   DATA[746,36] := 1.730048;
   DATA[746,37] := 189.9032;
   DATA[746,38] := 0.000128152;
   DATA[746,39] := 1.0;
   DATA[747,0] := 2.556449;
   DATA[747,1] := 537.959;
   DATA[747,2] := 2.0;
   DATA[747,3] := 1.0;
   DATA[747,4] := 262.1764;
   DATA[747,5] := 8.395475;
   DATA[747,6] := 327.5827;
   DATA[747,7] := 2.323647;
   DATA[747,9] := 1.0;
   DATA[747,10] := 1.0;
   DATA[747,11] := 2.016774;
   DATA[747,13] := 1002.908;
   DATA[747,14] := 1.0;
   DATA[747,15] := 1.0;
   DATA[747,16] := 1.0;
   DATA[747,17] := 1.0;
   DATA[747,18] := 1.0;
   DATA[747,19] := 1.0;
   DATA[747,20] := 148.808;
   DATA[747,21] := 155.8062;
   DATA[747,22] := 1.720309;
   DATA[747,23] := 993.899;
   DATA[747,24] := 2.0;
   DATA[747,25] := 2.0;
   DATA[747,26] := 7.878942;
   DATA[747,27] := 144.7321;
   DATA[747,28] := 263.1056;
   DATA[747,29] := 12.11228;
   DATA[747,30] := 1.731095;
   DATA[747,31] := 1.291789;
   DATA[747,32] := 0.7352687;
   DATA[747,33] := 0.3066329;
   DATA[747,34] := 2.0;
   DATA[747,35] := 251.2977;
   DATA[747,36] := 1.730048;
   DATA[747,37] := 190.0154;
   DATA[747,38] := 0.000128152;
   DATA[747,39] := 1.0;
   DATA[748,0] := 2.536912;
   DATA[748,1] := 538.1553;
   DATA[748,2] := 2.0;
   DATA[748,3] := 1.0;
   DATA[748,4] := 262.1764;
   DATA[748,5] := 8.399321;
   DATA[748,6] := 327.5827;
   DATA[748,7] := 2.09464;
   DATA[748,9] := 1.0;
   DATA[748,10] := 1.0;
   DATA[748,11] := 2.010372;
   DATA[748,13] := 1003.228;
   DATA[748,14] := 1.0;
   DATA[748,15] := 1.0;
   DATA[748,16] := 1.0;
   DATA[748,17] := 1.0;
   DATA[748,18] := 1.0;
   DATA[748,19] := 1.0;
   DATA[748,20] := 148.808;
   DATA[748,21] := 155.8062;
   DATA[748,22] := 1.72159;
   DATA[748,23] := 993.8221;
   DATA[748,24] := 2.0;
   DATA[748,25] := 2.0;
   DATA[748,26] := 7.878942;
   DATA[748,27] := 144.7321;
   DATA[748,28] := 263.1056;
   DATA[748,29] := 12.11228;
   DATA[748,30] := 1.731095;
   DATA[748,31] := 1.288971;
   DATA[748,32] := 0.7352687;
   DATA[748,33] := 0.3066329;
   DATA[748,34] := 2.0;
   DATA[748,35] := 251.2977;
   DATA[748,36] := 1.730048;
   DATA[748,37] := 190.0795;
   DATA[748,38] := 0.000128152;
   DATA[748,39] := 1.0;
   DATA[749,0] := 2.514813;
   DATA[749,1] := 538.5479;
   DATA[749,2] := 2.0;
   DATA[749,3] := 1.0;
   DATA[749,4] := 262.1764;
   DATA[749,5] := 8.399321;
   DATA[749,6] := 327.5827;
   DATA[749,7] := 1.782847;
   DATA[749,9] := 1.0;
   DATA[749,10] := 1.0;
   DATA[749,11] := 2.010372;
   DATA[749,13] := 1003.749;
   DATA[749,14] := 1.0;
   DATA[749,15] := 1.0;
   DATA[749,16] := 1.0;
   DATA[749,17] := 1.0;
   DATA[749,18] := 1.0;
   DATA[749,19] := 1.0;
   DATA[749,20] := 148.808;
   DATA[749,21] := 155.6524;
   DATA[749,22] := 1.721975;
   DATA[749,23] := 993.4376;
   DATA[749,24] := 2.0;
   DATA[749,25] := 2.0;
   DATA[749,26] := 7.878942;
   DATA[749,27] := 144.7321;
   DATA[749,28] := 263.1056;
   DATA[749,29] := 12.11228;
   DATA[749,30] := 1.731095;
   DATA[749,31] := 1.282951;
   DATA[749,32] := 0.7352687;
   DATA[749,33] := 0.3066329;
   DATA[749,34] := 2.0;
   DATA[749,35] := 251.2977;
   DATA[749,36] := 1.730048;
   DATA[749,37] := 190.0795;
   DATA[749,38] := 0.000128152;
   DATA[749,39] := 1.0;
   DATA[750,0] := 2.496237;
   DATA[750,1] := 538.8619;
   DATA[750,2] := 2.0;
   DATA[750,3] := 1.0;
   DATA[750,4] := 262.1764;
   DATA[750,5] := 8.399321;
   DATA[750,6] := 327.5827;
   DATA[750,7] := 1.39365;
   DATA[750,9] := 1.0;
   DATA[750,10] := 1.0;
   DATA[750,11] := 2.010372;
   DATA[750,13] := 1004.31;
   DATA[750,14] := 1.0;
   DATA[750,15] := 1.0;
   DATA[750,16] := 1.0;
   DATA[750,17] := 1.0;
   DATA[750,18] := 1.0;
   DATA[750,19] := 1.0;
   DATA[750,20] := 148.808;
   DATA[750,21] := 155.6524;
   DATA[750,22] := 1.72159;
   DATA[750,23] := 993.6683;
   DATA[750,24] := 2.0;
   DATA[750,25] := 2.0;
   DATA[750,26] := 7.878942;
   DATA[750,27] := 144.7321;
   DATA[750,28] := 263.1056;
   DATA[750,29] := 12.11228;
   DATA[750,30] := 1.731095;
   DATA[750,31] := 1.282439;
   DATA[750,32] := 0.7352687;
   DATA[750,33] := 0.3066329;
   DATA[750,34] := 2.0;
   DATA[750,35] := 251.2977;
   DATA[750,36] := 1.730048;
   DATA[750,37] := 190.0795;
   DATA[750,38] := 0.000128152;
   DATA[750,39] := 1.0;
   DATA[751,0] := 2.480223;
   DATA[751,1] := 538.8226;
   DATA[751,2] := 2.0;
   DATA[751,3] := 1.0;
   DATA[751,4] := 262.1764;
   DATA[751,5] := 8.399321;
   DATA[751,6] := 327.5827;
   DATA[751,7] := 1.022395;
   DATA[751,9] := 1.0;
   DATA[751,10] := 1.0;
   DATA[751,11] := 2.010372;
   DATA[751,13] := 1004.951;
   DATA[751,14] := 1.0;
   DATA[751,15] := 1.0;
   DATA[751,16] := 1.0;
   DATA[751,17] := 1.0;
   DATA[751,18] := 1.0;
   DATA[751,19] := 1.0;
   DATA[751,20] := 148.808;
   DATA[751,21] := 155.6524;
   DATA[751,22] := 1.719668;
   DATA[751,23] := 993.1684;
   DATA[751,24] := 2.0;
   DATA[751,25] := 2.0;
   DATA[751,26] := 7.878942;
   DATA[751,27] := 144.7321;
   DATA[751,28] := 263.1056;
   DATA[751,29] := 12.11228;
   DATA[751,30] := 1.731735;
   DATA[751,31] := 1.281927;
   DATA[751,32] := 0.7352687;
   DATA[751,33] := 0.3066329;
   DATA[751,34] := 2.0;
   DATA[751,35] := 251.2977;
   DATA[751,36] := 1.762086;
   DATA[751,37] := 190.0795;
   DATA[751,38] := 0.000128152;
   DATA[751,39] := 1.0;
   DATA[752,0] := 2.464849;
   DATA[752,1] := 538.9796;
   DATA[752,2] := 2.0;
   DATA[752,3] := 1.0;
   DATA[752,4] := 262.1764;
   DATA[752,5] := 8.399321;
   DATA[752,6] := 327.3263;
   DATA[752,7] := 0.6416557;
   DATA[752,9] := 1.0;
   DATA[752,10] := 1.0;
   DATA[752,11] := 2.010372;
   DATA[752,13] := 1005.351;
   DATA[752,14] := 1.0;
   DATA[752,15] := 1.0;
   DATA[752,16] := 1.0;
   DATA[752,17] := 1.0;
   DATA[752,18] := 1.0;
   DATA[752,19] := 1.0;
   DATA[752,20] := 148.808;
   DATA[752,21] := 155.6524;
   DATA[752,22] := 1.719668;
   DATA[752,23] := 993.1299;
   DATA[752,24] := 2.0;
   DATA[752,25] := 2.0;
   DATA[752,26] := 7.878942;
   DATA[752,27] := 144.7321;
   DATA[752,28] := 263.1056;
   DATA[752,29] := 12.11228;
   DATA[752,30] := 1.734427;
   DATA[752,31] := 1.288075;
   DATA[752,32] := 0.7352687;
   DATA[752,33] := 0.3066329;
   DATA[752,34] := 2.0;
   DATA[752,35] := 251.2977;
   DATA[752,36] := 1.762086;
   DATA[752,37] := 190.0795;
   DATA[752,38] := 0.000128152;
   DATA[752,39] := 1.0;
   DATA[753,0] := 2.449156;
   DATA[753,1] := 539.1759;
   DATA[753,2] := 2.0;
   DATA[753,3] := 1.0;
   DATA[753,4] := 262.1764;
   DATA[753,5] := 8.399321;
   DATA[753,6] := 326.9931;
   DATA[753,7] := 0.3813795;
   DATA[753,8] := 1.0;
   DATA[753,9] := 1.0;
   DATA[753,10] := 1.0;
   DATA[753,11] := 2.010372;
   DATA[753,13] := 1006.272;
   DATA[753,14] := 1.0;
   DATA[753,15] := 1.0;
   DATA[753,16] := 1.0;
   DATA[753,17] := 1.0;
   DATA[753,18] := 1.0;
   DATA[753,19] := 1.0;
   DATA[753,20] := 148.808;
   DATA[753,21] := 155.6524;
   DATA[753,22] := 1.721719;
   DATA[753,23] := 992.361;
   DATA[753,24] := 2.0;
   DATA[753,25] := 2.0;
   DATA[753,26] := 7.878942;
   DATA[753,27] := 144.7321;
   DATA[753,28] := 263.1056;
   DATA[753,29] := 12.11228;
   DATA[753,30] := 1.734427;
   DATA[753,31] := 1.291277;
   DATA[753,32] := 0.7352687;
   DATA[753,33] := 0.3066329;
   DATA[753,34] := 2.0;
   DATA[753,35] := 251.2977;
   DATA[753,36] := 1.762086;
   DATA[753,37] := 190.0795;
   DATA[753,38] := 0.000128152;
   DATA[753,39] := 1.0;
   DATA[754,0] := 2.433462;
   DATA[754,1] := 539.7646;
   DATA[754,2] := 2.0;
   DATA[754,3] := 1.0;
   DATA[754,4] := 262.1764;
   DATA[754,5] := 8.399321;
   DATA[754,6] := 326.7111;
   DATA[754,7] := 0.2296479;
   DATA[754,8] := 1.0;
   DATA[754,9] := 1.0;
   DATA[754,10] := 1.0;
   DATA[754,11] := 2.010372;
   DATA[754,13] := 1006.753;
   DATA[754,14] := 1.0;
   DATA[754,15] := 1.0;
   DATA[754,16] := 1.0;
   DATA[754,17] := 1.0;
   DATA[754,18] := 1.0;
   DATA[754,19] := 1.0;
   DATA[754,20] := 148.808;
   DATA[754,21] := 155.4473;
   DATA[754,22] := 1.721719;
   DATA[754,23] := 992.3225;
   DATA[754,24] := 2.0;
   DATA[754,25] := 2.0;
   DATA[754,26] := 7.878942;
   DATA[754,27] := 144.7321;
   DATA[754,28] := 263.1056;
   DATA[754,29] := 12.11228;
   DATA[754,30] := 1.734427;
   DATA[754,31] := 1.291405;
   DATA[754,32] := 0.7352687;
   DATA[754,33] := 0.3066329;
   DATA[754,34] := 2.0;
   DATA[754,35] := 251.2977;
   DATA[754,36] := 1.762086;
   DATA[754,37] := 190.0795;
   DATA[754,38] := 0.000128152;
   DATA[754,39] := 1.0;
   DATA[755,0] := 2.423213;
   DATA[755,1] := 539.804;
   DATA[755,2] := 2.0;
   DATA[755,3] := 1.0;
   DATA[755,4] := 262.1764;
   DATA[755,5] := 8.399321;
   DATA[755,6] := 326.7111;
   DATA[755,7] := 0.1289206;
   DATA[755,8] := 1.0;
   DATA[755,9] := 1.0;
   DATA[755,10] := 1.0;
   DATA[755,11] := 2.010372;
   DATA[755,13] := 1006.953;
   DATA[755,14] := 1.0;
   DATA[755,15] := 1.0;
   DATA[755,16] := 1.0;
   DATA[755,17] := 1.0;
   DATA[755,18] := 1.0;
   DATA[755,19] := 1.0;
   DATA[755,20] := 148.808;
   DATA[755,21] := 155.4217;
   DATA[755,22] := 1.721719;
   DATA[755,23] := 991.5535;
   DATA[755,24] := 2.0;
   DATA[755,25] := 2.0;
   DATA[755,26] := 7.878942;
   DATA[755,27] := 144.8603;
   DATA[755,28] := 263.1056;
   DATA[755,29] := 12.11228;
   DATA[755,30] := 1.733786;
   DATA[755,31] := 1.291405;
   DATA[755,32] := 0.7352687;
   DATA[755,33] := 0.3066329;
   DATA[755,34] := 2.0;
   DATA[755,35] := 251.2977;
   DATA[755,36] := 1.762086;
   DATA[755,37] := 190.0154;
   DATA[755,38] := 0.000128152;
   DATA[755,39] := 1.0;
   DATA[756,0] := 2.41905;
   DATA[756,1] := 540.3535;
   DATA[756,2] := 2.0;
   DATA[756,3] := 1.0;
   DATA[756,4] := 262.1764;
   DATA[756,5] := 8.399321;
   DATA[756,6] := 326.5573;
   DATA[756,7] := 0.070099;
   DATA[756,8] := 1.0;
   DATA[756,9] := 1.0;
   DATA[756,10] := 1.0;
   DATA[756,11] := 2.010372;
   DATA[756,13] := 1007.474;
   DATA[756,14] := 1.0;
   DATA[756,15] := 1.0;
   DATA[756,16] := 1.0;
   DATA[756,17] := 1.0;
   DATA[756,18] := 1.0;
   DATA[756,19] := 1.0;
   DATA[756,20] := 148.808;
   DATA[756,21] := 155.4217;
   DATA[756,22] := 1.720053;
   DATA[756,23] := 991.7457;
   DATA[756,24] := 2.0;
   DATA[756,25] := 2.0;
   DATA[756,26] := 7.878942;
   DATA[756,27] := 144.8603;
   DATA[756,28] := 263.1056;
   DATA[756,29] := 12.11228;
   DATA[756,30] := 1.731223;
   DATA[756,31] := 1.29243;
   DATA[756,32] := 0.7352687;
   DATA[756,33] := 0.3066329;
   DATA[756,34] := 2.0;
   DATA[756,35] := 251.2977;
   DATA[756,36] := 1.762086;
   DATA[756,37] := 189.8872;
   DATA[756,38] := 0.000128152;
   DATA[756,39] := 1.0;
   DATA[757,0] := 2.41905;
   DATA[757,1] := 540.5497;
   DATA[757,2] := 2.0;
   DATA[757,3] := 1.0;
   DATA[757,4] := 262.1764;
   DATA[757,5] := 8.401243;
   DATA[757,6] := 325.9677;
   DATA[757,7] := 0.03575433;
   DATA[757,8] := 1.0;
   DATA[757,9] := 1.0;
   DATA[757,10] := 1.0;
   DATA[757,11] := 2.010372;
   DATA[757,13] := 1007.835;
   DATA[757,14] := 1.0;
   DATA[757,15] := 1.0;
   DATA[757,16] := 1.0;
   DATA[757,17] := 1.0;
   DATA[757,18] := 1.0;
   DATA[757,19] := 1.0;
   DATA[757,20] := 148.808;
   DATA[757,21] := 155.4217;
   DATA[757,22] := 1.719668;
   DATA[757,23] := 991.3997;
   DATA[757,24] := 2.0;
   DATA[757,25] := 2.0;
   DATA[757,26] := 7.878942;
   DATA[757,27] := 144.8603;
   DATA[757,28] := 263.1056;
   DATA[757,29] := 12.11228;
   DATA[757,30] := 1.731223;
   DATA[757,31] := 1.302165;
   DATA[757,32] := 0.7352687;
   DATA[757,33] := 0.3066329;
   DATA[757,34] := 2.0;
   DATA[757,35] := 251.1535;
   DATA[757,36] := 1.762086;
   DATA[757,37] := 189.8552;
   DATA[757,38] := 0.000128152;
   DATA[757,39] := 1.0;
   DATA[758,0] := 2.437626;
   DATA[758,1] := 541.0992;
   DATA[758,2] := 2.0;
   DATA[758,3] := 1.0;
   DATA[758,4] := 262.1764;
   DATA[758,5] := 8.401243;
   DATA[758,6] := 325.4294;
   DATA[758,7] := 0.01435299;
   DATA[758,8] := 1.0;
   DATA[758,9] := 1.0;
   DATA[758,10] := 1.0;
   DATA[758,11] := 2.010372;
   DATA[758,13] := 1008.355;
   DATA[758,14] := 1.0;
   DATA[758,15] := 1.0;
   DATA[758,16] := 1.0;
   DATA[758,17] := 1.0;
   DATA[758,18] := 1.0;
   DATA[758,19] := 1.0;
   DATA[758,20] := 148.808;
   DATA[758,21] := 155.4217;
   DATA[758,22] := 1.719668;
   DATA[758,23] := 991.3228;
   DATA[758,24] := 2.0;
   DATA[758,25] := 2.0;
   DATA[758,26] := 7.878942;
   DATA[758,27] := 144.8603;
   DATA[758,28] := 263.1056;
   DATA[758,29] := 12.11228;
   DATA[758,30] := 1.731223;
   DATA[758,31] := 1.311387;
   DATA[758,32] := 0.7352687;
   DATA[758,33] := 0.3066329;
   DATA[758,34] := 2.0;
   DATA[758,35] := 251.1055;
   DATA[758,36] := 1.762086;
   DATA[758,37] := 189.8552;
   DATA[758,38] := 0.000128152;
   DATA[758,39] := 1.0;
   DATA[759,0] := 2.461006;
   DATA[759,1] := 540.8245;
   DATA[759,2] := 2.0;
   DATA[759,3] := 1.0;
   DATA[759,4] := 262.1764;
   DATA[759,5] := 8.405088;
   DATA[759,6] := 325.4294;
   DATA[759,7] := 0.000512607;
   DATA[759,8] := 1.0;
   DATA[759,9] := 1.0;
   DATA[759,10] := 1.0;
   DATA[759,11] := 2.010372;
   DATA[759,13] := 1008.275;
   DATA[759,14] := 1.0;
   DATA[759,15] := 1.0;
   DATA[759,16] := 1.0;
   DATA[759,17] := 1.0;
   DATA[759,18] := 1.0;
   DATA[759,19] := 1.0;
   DATA[759,20] := 148.808;
   DATA[759,21] := 155.5242;
   DATA[759,22] := 1.719668;
   DATA[759,23] := 990.4768;
   DATA[759,24] := 2.0;
   DATA[759,25] := 2.0;
   DATA[759,26] := 7.878942;
   DATA[759,27] := 144.8603;
   DATA[759,28] := 263.1056;
   DATA[759,29] := 12.11228;
   DATA[759,30] := 1.731223;
   DATA[759,31] := 1.306648;
   DATA[759,32] := 0.7352687;
   DATA[759,33] := 0.3066329;
   DATA[759,34] := 2.0;
   DATA[759,35] := 251.0734;
   DATA[759,36] := 1.746067;
   DATA[759,37] := 189.8231;
   DATA[759,38] := 0.000128152;
   DATA[759,39] := 1.0;
   DATA[760,0] := 2.478621;
   DATA[760,1] := 541.4918;
   DATA[760,2] := 2.0;
   DATA[760,3] := 1.0;
   DATA[760,4] := 262.1764;
   DATA[760,5] := 8.40605;
   DATA[760,6] := 324.7885;
   DATA[760,7] := 0.000512607;
   DATA[760,8] := 1.0;
   DATA[760,9] := 1.0;
   DATA[760,10] := 1.0;
   DATA[760,11] := 2.010372;
   DATA[760,13] := 1008.355;
   DATA[760,14] := 1.0;
   DATA[760,15] := 1.0;
   DATA[760,16] := 1.0;
   DATA[760,17] := 1.0;
   DATA[760,18] := 1.0;
   DATA[760,19] := 1.0;
   DATA[760,20] := 148.808;
   DATA[760,21] := 155.5242;
   DATA[760,22] := 1.719924;
   DATA[760,23] := 990.3999;
   DATA[760,24] := 2.0;
   DATA[760,25] := 2.0;
   DATA[760,26] := 7.878942;
   DATA[760,27] := 144.8603;
   DATA[760,28] := 263.1056;
   DATA[760,29] := 11.95847;
   DATA[760,30] := 1.731223;
   DATA[760,31] := 1.308185;
   DATA[760,32] := 0.7352687;
   DATA[760,33] := 0.3066329;
   DATA[760,34] := 2.0;
   DATA[760,35] := 250.8652;
   DATA[760,36] := 1.746067;
   DATA[760,37] := 189.727;
   DATA[760,38] := 0.000128152;
   DATA[760,39] := 1.0;
   DATA[761,0] := 2.502642;
   DATA[761,1] := 542.0021;
   DATA[761,2] := 2.0;
   DATA[761,3] := 1.0;
   DATA[761,4] := 262.1764;
   DATA[761,5] := 8.40605;
   DATA[761,6] := 324.1989;
   DATA[761,7] := 0.000512607;
   DATA[761,8] := 1.0;
   DATA[761,9] := 1.0;
   DATA[761,10] := 1.0;
   DATA[761,11] := 2.010372;
   DATA[761,13] := 1008.636;
   DATA[761,14] := 1.0;
   DATA[761,15] := 1.0;
   DATA[761,16] := 1.0;
   DATA[761,17] := 1.0;
   DATA[761,18] := 1.0;
   DATA[761,19] := 1.0;
   DATA[761,20] := 148.808;
   DATA[761,21] := 155.5242;
   DATA[761,22] := 1.719924;
   DATA[761,23] := 990.0154;
   DATA[761,24] := 2.0;
   DATA[761,25] := 2.0;
   DATA[761,26] := 7.878942;
   DATA[761,27] := 144.8603;
   DATA[761,28] := 263.1056;
   DATA[761,29] := 11.95847;
   DATA[761,30] := 1.731223;
   DATA[761,31] := 1.3119;
   DATA[761,32] := 0.7352687;
   DATA[761,33] := 0.3066329;
   DATA[761,34] := 2.0;
   DATA[761,35] := 250.8652;
   DATA[761,36] := 1.746067;
   DATA[761,37] := 189.727;
   DATA[761,38] := 0.000128152;
   DATA[761,39] := 1.0;
   DATA[762,0] := 2.515453;
   DATA[762,1] := 542.3553;
   DATA[762,2] := 2.0;
   DATA[762,3] := 1.0;
   DATA[762,4] := 262.1764;
   DATA[762,5] := 8.408293;
   DATA[762,6] := 323.7375;
   DATA[762,7] := 0.000512607;
   DATA[762,8] := 1.0;
   DATA[762,9] := 1.0;
   DATA[762,10] := 1.0;
   DATA[762,11] := 2.035982;
   DATA[762,13] := 1008.475;
   DATA[762,14] := 1.0;
   DATA[762,15] := 1.0;
   DATA[762,16] := 1.0;
   DATA[762,17] := 1.0;
   DATA[762,18] := 1.0;
   DATA[762,19] := 1.0;
   DATA[762,20] := 148.808;
   DATA[762,21] := 155.5242;
   DATA[762,22] := 1.719924;
   DATA[762,23] := 989.8231;
   DATA[762,24] := 2.0;
   DATA[762,25] := 2.0;
   DATA[762,26] := 7.878942;
   DATA[762,27] := 144.8603;
   DATA[762,28] := 263.1056;
   DATA[762,29] := 11.95847;
   DATA[762,30] := 1.731223;
   DATA[762,31] := 1.304855;
   DATA[762,32] := 0.7352687;
   DATA[762,33] := 0.3066329;
   DATA[762,34] := 2.0;
   DATA[762,35] := 250.8652;
   DATA[762,36] := 1.746067;
   DATA[762,37] := 189.6629;
   DATA[762,38] := 0.000128152;
   DATA[762,39] := 1.0;
   DATA[763,0] := 2.528264;
   DATA[763,1] := 542.9442;
   DATA[763,2] := 2.0;
   DATA[763,3] := 1.0;
   DATA[763,4] := 262.1764;
   DATA[763,5] := 8.412458;
   DATA[763,6] := 323.3017;
   DATA[763,7] := 0.000512607;
   DATA[763,8] := 1.0;
   DATA[763,9] := 1.0;
   DATA[763,10] := 1.0;
   DATA[763,11] := 2.035982;
   DATA[763,13] := 1008.876;
   DATA[763,14] := 1.0;
   DATA[763,15] := 1.0;
   DATA[763,16] := 1.0;
   DATA[763,17] := 1.0;
   DATA[763,18] := 1.0;
   DATA[763,19] := 1.0;
   DATA[763,20] := 148.808;
   DATA[763,21] := 155.5242;
   DATA[763,22] := 1.719924;
   DATA[763,23] := 989.5155;
   DATA[763,24] := 2.0;
   DATA[763,25] := 2.0;
   DATA[763,26] := 7.878942;
   DATA[763,27] := 144.8603;
   DATA[763,28] := 263.1056;
   DATA[763,29] := 11.95847;
   DATA[763,30] := 1.731095;
   DATA[763,31] := 1.291789;
   DATA[763,32] := 0.7352687;
   DATA[763,33] := 0.3066329;
   DATA[763,34] := 2.0;
   DATA[763,35] := 250.8652;
   DATA[763,36] := 1.537821;
   DATA[763,37] := 189.6629;
   DATA[763,38] := 0.000128152;
   DATA[763,39] := 1.0;
   DATA[764,0] := 2.533068;
   DATA[764,1] := 543.4937;
   DATA[764,2] := 2.0;
   DATA[764,3] := 1.0;
   DATA[764,4] := 262.1764;
   DATA[764,5] := 8.412458;
   DATA[764,6] := 323.0197;
   DATA[764,7] := 0.000512607;
   DATA[764,8] := 1.0;
   DATA[764,9] := 1.0;
   DATA[764,10] := 1.0;
   DATA[764,11] := 2.026378;
   DATA[764,13] := 1008.836;
   DATA[764,14] := 1.0;
   DATA[764,15] := 1.0;
   DATA[764,16] := 1.0;
   DATA[764,17] := 1.0;
   DATA[764,18] := 1.0;
   DATA[764,19] := 1.0;
   DATA[764,20] := 148.808;
   DATA[764,21] := 155.5242;
   DATA[764,22] := 1.718771;
   DATA[764,23] := 989.4001;
   DATA[764,24] := 2.0;
   DATA[764,25] := 2.0;
   DATA[764,26] := 7.878942;
   DATA[764,27] := 144.8603;
   DATA[764,28] := 263.1056;
   DATA[764,29] := 11.95847;
   DATA[764,30] := 1.730838;
   DATA[764,31] := 1.28167;
   DATA[764,32] := 0.7352687;
   DATA[764,33] := 0.3066329;
   DATA[764,34] := 2.0;
   DATA[764,35] := 250.8652;
   DATA[764,36] := 1.537821;
   DATA[764,37] := 189.6629;
   DATA[764,38] := 0.000128152;
   DATA[764,39] := 1.0;
   DATA[765,0] := 2.533068;
   DATA[765,1] := 544.0432;
   DATA[765,2] := 2.0;
   DATA[765,3] := 1.0;
   DATA[765,4] := 262.1764;
   DATA[765,5] := 8.412458;
   DATA[765,6] := 322.6096;
   DATA[765,7] := 0.000512607;
   DATA[765,8] := 1.0;
   DATA[765,9] := 1.0;
   DATA[765,10] := 1.0;
   DATA[765,11] := 2.013573;
   DATA[765,13] := 1009.076;
   DATA[765,14] := 1.0;
   DATA[765,15] := 1.0;
   DATA[765,16] := 1.0;
   DATA[765,17] := 1.0;
   DATA[765,18] := 1.0;
   DATA[765,19] := 1.0;
   DATA[765,20] := 148.808;
   DATA[765,21] := 155.5242;
   DATA[765,22] := 1.717233;
   DATA[765,23] := 989.3232;
   DATA[765,24] := 2.0;
   DATA[765,25] := 2.0;
   DATA[765,26] := 7.878942;
   DATA[765,27] := 144.8603;
   DATA[765,28] := 263.1056;
   DATA[765,29] := 11.95847;
   DATA[765,30] := 1.730069;
   DATA[765,31] := 1.28167;
   DATA[765,32] := 0.7352687;
   DATA[765,33] := 0.3066329;
   DATA[765,34] := 2.0;
   DATA[765,35] := 250.8652;
   DATA[765,36] := 1.665972;
   DATA[765,37] := 189.5828;
   DATA[765,38] := 0.000128152;
   DATA[765,39] := 1.0;
   DATA[766,0] := 2.533068;
   DATA[766,1] := 544.7498;
   DATA[766,2] := 2.0;
   DATA[766,3] := 1.0;
   DATA[766,4] := 262.1764;
   DATA[766,5] := 8.417906;
   DATA[766,6] := 321.8405;
   DATA[766,7] := 0.000512607;
   DATA[766,8] := 1.0;
   DATA[766,9] := 1.0;
   DATA[766,10] := 1.0;
   DATA[766,11] := 2.013573;
   DATA[766,13] := 1008.916;
   DATA[766,14] := 1.0;
   DATA[766,15] := 1.0;
   DATA[766,16] := 1.0;
   DATA[766,17] := 1.0;
   DATA[766,18] := 1.0;
   DATA[766,19] := 1.0;
   DATA[766,20] := 148.808;
   DATA[766,21] := 155.5242;
   DATA[766,22] := 1.717233;
   DATA[766,23] := 989.2848;
   DATA[766,24] := 2.0;
   DATA[766,25] := 2.0;
   DATA[766,26] := 7.878942;
   DATA[766,27] := 144.8603;
   DATA[766,28] := 263.1056;
   DATA[766,29] := 11.95847;
   DATA[766,30] := 1.728275;
   DATA[766,31] := 1.28167;
   DATA[766,32] := 0.7352687;
   DATA[766,33] := 0.3066329;
   DATA[766,34] := 2.0;
   DATA[766,35] := 250.8652;
   DATA[766,36] := 1.69801;
   DATA[766,37] := 189.5828;
   DATA[766,38] := 0.000128152;
   DATA[766,39] := 1.0;
   DATA[767,0] := 2.531467;
   DATA[767,1] := 545.4563;
   DATA[767,2] := 2.0;
   DATA[767,3] := 1.0;
   DATA[767,4] := 262.1764;
   DATA[767,5] := 8.422392;
   DATA[767,6] := 321.4048;
   DATA[767,8] := 1.0;
   DATA[767,9] := 1.0;
   DATA[767,10] := 1.0;
   DATA[767,11] := 2.013573;
   DATA[767,13] := 1009.637;
   DATA[767,14] := 1.0;
   DATA[767,15] := 1.0;
   DATA[767,16] := 1.0;
   DATA[767,17] := 1.0;
   DATA[767,18] := 1.0;
   DATA[767,19] := 1.0;
   DATA[767,20] := 148.808;
   DATA[767,21] := 155.5242;
   DATA[767,22] := 1.717233;
   DATA[767,23] := 988.5157;
   DATA[767,24] := 2.0;
   DATA[767,25] := 2.0;
   DATA[767,26] := 7.878942;
   DATA[767,27] := 144.8603;
   DATA[767,28] := 263.1056;
   DATA[767,29] := 11.95847;
   DATA[767,30] := 1.728275;
   DATA[767,31] := 1.294479;
   DATA[767,32] := 0.7352687;
   DATA[767,33] := 0.3066329;
   DATA[767,34] := 2.0;
   DATA[767,35] := 250.7049;
   DATA[767,36] := 1.69801;
   DATA[767,37] := 189.4066;
   DATA[767,38] := 0.000128152;
   DATA[767,39] := 1.0;
   DATA[768,0] := 2.531467;
   DATA[768,1] := 546.3199;
   DATA[768,2] := 2.0;
   DATA[768,3] := 1.0;
   DATA[768,4] := 262.1764;
   DATA[768,5] := 8.422712;
   DATA[768,6] := 320.8665;
   DATA[768,8] := 1.0;
   DATA[768,9] := 1.0;
   DATA[768,10] := 1.0;
   DATA[768,11] := 2.013573;
   DATA[768,13] := 1009.637;
   DATA[768,14] := 1.0;
   DATA[768,15] := 1.0;
   DATA[768,16] := 1.0;
   DATA[768,17] := 1.0;
   DATA[768,18] := 1.0;
   DATA[768,19] := 1.0;
   DATA[768,20] := 148.808;
   DATA[768,21] := 155.5242;
   DATA[768,22] := 1.717233;
   DATA[768,23] := 988.0543;
   DATA[768,24] := 2.0;
   DATA[768,25] := 2.0;
   DATA[768,26] := 7.878942;
   DATA[768,27] := 144.8603;
   DATA[768,28] := 263.1056;
   DATA[768,29] := 11.95847;
   DATA[768,30] := 1.728275;
   DATA[768,31] := 1.294479;
   DATA[768,32] := 0.7352687;
   DATA[768,33] := 0.3066329;
   DATA[768,34] := 2.0;
   DATA[768,35] := 250.6248;
   DATA[768,36] := 1.69801;
   DATA[768,37] := 189.3265;
   DATA[768,38] := 0.000128152;
   DATA[768,39] := 1.0;
   DATA[769,0] := 2.531467;
   DATA[769,1] := 546.4376;
   DATA[769,2] := 2.0;
   DATA[769,3] := 1.0;
   DATA[769,4] := 262.1764;
   DATA[769,5] := 8.425276;
   DATA[769,6] := 320.687;
   DATA[769,8] := 1.0;
   DATA[769,9] := 1.0;
   DATA[769,10] := 1.0;
   DATA[769,11] := 2.013573;
   DATA[769,13] := 1009.917;
   DATA[769,14] := 1.0;
   DATA[769,15] := 1.0;
   DATA[769,16] := 1.0;
   DATA[769,17] := 1.0;
   DATA[769,18] := 1.0;
   DATA[769,19] := 1.0;
   DATA[769,20] := 148.808;
   DATA[769,21] := 155.5242;
   DATA[769,22] := 1.717233;
   DATA[769,23] := 987.5544;
   DATA[769,24] := 2.0;
   DATA[769,25] := 2.0;
   DATA[769,26] := 7.878942;
   DATA[769,27] := 144.9116;
   DATA[769,28] := 263.1056;
   DATA[769,29] := 11.95847;
   DATA[769,30] := 1.728275;
   DATA[769,31] := 1.291533;
   DATA[769,32] := 0.7352687;
   DATA[769,33] := 0.3074016;
   DATA[769,34] := 2.0;
   DATA[769,35] := 250.6248;
   DATA[769,36] := 1.69801;
   DATA[769,37] := 189.3265;
   DATA[769,38] := 0.000128152;
   DATA[769,39] := 1.0;
   DATA[770,0] := 2.53435;
   DATA[770,1] := 546.6732;
   DATA[770,2] := 2.0;
   DATA[770,3] := 1.0;
   DATA[770,4] := 262.1764;
   DATA[770,5] := 8.432005;
   DATA[770,6] := 320.2512;
   DATA[770,8] := 1.0;
   DATA[770,9] := 1.0;
   DATA[770,10] := 1.0;
   DATA[770,11] := 2.013573;
   DATA[770,13] := 1009.877;
   DATA[770,14] := 1.0;
   DATA[770,15] := 1.0;
   DATA[770,16] := 1.0;
   DATA[770,17] := 1.0;
   DATA[770,18] := 1.0;
   DATA[770,19] := 1.0;
   DATA[770,20] := 148.808;
   DATA[770,21] := 155.5242;
   DATA[770,22] := 1.715952;
   DATA[770,23] := 987.1315;
   DATA[770,24] := 2.0;
   DATA[770,25] := 2.0;
   DATA[770,26] := 7.878942;
   DATA[770,27] := 144.9628;
   DATA[770,28] := 263.1056;
   DATA[770,29] := 11.95847;
   DATA[770,30] := 1.728275;
   DATA[770,31] := 1.290765;
   DATA[770,32] := 0.7352687;
   DATA[770,33] := 0.3074016;
   DATA[770,34] := 2.0;
   DATA[770,35] := 250.785;
   DATA[770,36] := 1.69801;
   DATA[770,37] := 189.5027;
   DATA[770,38] := 0.000128152;
   DATA[770,39] := 1.0;
   DATA[771,0] := 2.53435;
   DATA[771,1] := 546.6732;
   DATA[771,2] := 2.0;
   DATA[771,3] := 1.0;
   DATA[771,4] := 262.1764;
   DATA[771,5] := 8.432005;
   DATA[771,6] := 320.2512;
   DATA[771,8] := 1.0;
   DATA[771,9] := 1.0;
   DATA[771,10] := 1.0;
   DATA[771,11] := 2.013573;
   DATA[771,13] := 1009.877;
   DATA[771,14] := 1.0;
   DATA[771,15] := 1.0;
   DATA[771,16] := 1.0;
   DATA[771,17] := 1.0;
   DATA[771,18] := 1.0;
   DATA[771,19] := 1.0;
   DATA[771,20] := 148.808;
   DATA[771,21] := 155.5242;
   DATA[771,22] := 1.715952;
   DATA[771,23] := 987.1315;
   DATA[771,24] := 2.0;
   DATA[771,25] := 2.0;
   DATA[771,26] := 7.878942;
   DATA[771,27] := 144.9628;
   DATA[771,28] := 263.1056;
   DATA[771,29] := 11.95847;
   DATA[771,30] := 1.728275;
   DATA[771,31] := 1.290765;
   DATA[771,32] := 0.7352687;
   DATA[771,33] := 0.3074016;
   DATA[771,34] := 2.0;
   DATA[771,35] := 250.785;
   DATA[771,36] := 1.69801;
   DATA[771,37] := 189.5027;
   DATA[771,38] := 0.000128152;
   DATA[771,39] := 1.0;
   DATA[772,0] := 2.537232;
   DATA[772,1] := 546.5947;
   DATA[772,2] := 2.0;
   DATA[772,3] := 1.0;
   DATA[772,4] := 262.1764;
   DATA[772,5] := 8.432005;
   DATA[772,6] := 319.5847;
   DATA[772,8] := 1.0;
   DATA[772,9] := 1.0;
   DATA[772,10] := 1.0;
   DATA[772,11] := 2.013573;
   DATA[772,13] := 1010.038;
   DATA[772,14] := 1.0;
   DATA[772,15] := 1.0;
   DATA[772,16] := 1.0;
   DATA[772,17] := 1.0;
   DATA[772,18] := 1.0;
   DATA[772,19] := 1.0;
   DATA[772,20] := 148.808;
   DATA[772,21] := 155.5242;
   DATA[772,22] := 1.715952;
   DATA[772,23] := 986.747;
   DATA[772,24] := 2.0;
   DATA[772,25] := 2.0;
   DATA[772,26] := 7.878942;
   DATA[772,27] := 144.9628;
   DATA[772,28] := 263.1056;
   DATA[772,29] := 11.95847;
   DATA[772,30] := 1.728275;
   DATA[772,31] := 1.282183;
   DATA[772,32] := 0.7352687;
   DATA[772,33] := 0.3074016;
   DATA[772,34] := 2.0;
   DATA[772,35] := 250.9613;
   DATA[772,36] := 1.69801;
   DATA[772,37] := 189.6949;
   DATA[772,38] := 0.000128152;
   DATA[772,39] := 1.0;
   DATA[773,0] := 2.537232;
   DATA[773,1] := 546.6339;
   DATA[773,2] := 2.0;
   DATA[773,3] := 1.0;
   DATA[773,4] := 262.1764;
   DATA[773,5] := 8.434568;
   DATA[773,6] := 319.5847;
   DATA[773,8] := 1.0;
   DATA[773,9] := 1.0;
   DATA[773,10] := 1.0;
   DATA[773,11] := 2.013573;
   DATA[773,13] := 1009.917;
   DATA[773,14] := 1.0;
   DATA[773,15] := 1.0;
   DATA[773,16] := 1.0;
   DATA[773,17] := 1.0;
   DATA[773,18] := 1.0;
   DATA[773,19] := 1.0;
   DATA[773,20] := 148.808;
   DATA[773,21] := 155.5242;
   DATA[773,22] := 1.715952;
   DATA[773,23] := 986.2087;
   DATA[773,24] := 2.0;
   DATA[773,25] := 2.0;
   DATA[773,26] := 7.878942;
   DATA[773,27] := 144.9628;
   DATA[773,28] := 263.1056;
   DATA[773,29] := 11.95847;
   DATA[773,30] := 1.728788;
   DATA[773,31] := 1.290252;
   DATA[773,32] := 0.7352687;
   DATA[773,33] := 0.3065048;
   DATA[773,34] := 2.0;
   DATA[773,35] := 250.9613;
   DATA[773,36] := 1.649953;
   DATA[773,37] := 189.759;
   DATA[773,38] := 0.000128152;
   DATA[773,39] := 1.0;
   DATA[774,0] := 2.537232;
   DATA[774,1] := 547.0264;
   DATA[774,2] := 2.0;
   DATA[774,3] := 1.0;
   DATA[774,4] := 262.1764;
   DATA[774,5] := 8.439695;
   DATA[774,6] := 318.9695;
   DATA[774,8] := 1.0;
   DATA[774,9] := 1.0;
   DATA[774,10] := 1.0;
   DATA[774,11] := 2.013573;
   DATA[774,13] := 1009.757;
   DATA[774,14] := 1.0;
   DATA[774,15] := 1.0;
   DATA[774,16] := 1.0;
   DATA[774,17] := 1.0;
   DATA[774,18] := 1.0;
   DATA[774,19] := 1.0;
   DATA[774,20] := 148.808;
   DATA[774,21] := 155.6524;
   DATA[774,22] := 1.717746;
   DATA[774,23] := 986.0164;
   DATA[774,24] := 2.0;
   DATA[774,25] := 2.0;
   DATA[774,26] := 7.878942;
   DATA[774,27] := 144.9628;
   DATA[774,28] := 263.1056;
   DATA[774,29] := 11.95847;
   DATA[774,30] := 1.731864;
   DATA[774,31] := 1.297554;
   DATA[774,32] := 0.7352687;
   DATA[774,33] := 0.3065048;
   DATA[774,34] := 2.0;
   DATA[774,35] := 250.9613;
   DATA[774,36] := 1.649953;
   DATA[774,37] := 189.759;
   DATA[774,38] := 0.000128152;
   DATA[774,39] := 1.0;
   DATA[775,0] := 2.537232;
   DATA[775,1] := 546.9872;
   DATA[775,2] := 2.0;
   DATA[775,3] := 1.0;
   DATA[775,4] := 262.1764;
   DATA[775,5] := 8.4429;
   DATA[775,6] := 318.9695;
   DATA[775,8] := 1.0;
   DATA[775,9] := 1.0;
   DATA[775,10] := 1.0;
   DATA[775,11] := 2.013573;
   DATA[775,13] := 1010.078;
   DATA[775,14] := 1.0;
   DATA[775,15] := 1.0;
   DATA[775,16] := 1.0;
   DATA[775,17] := 1.0;
   DATA[775,18] := 1.0;
   DATA[775,19] := 1.0;
   DATA[775,20] := 148.808;
   DATA[775,21] := 155.6524;
   DATA[775,22] := 1.717746;
   DATA[775,23] := 985.5934;
   DATA[775,24] := 2.0;
   DATA[775,25] := 2.0;
   DATA[775,26] := 7.878942;
   DATA[775,27] := 144.9628;
   DATA[775,28] := 263.1056;
   DATA[775,29] := 11.95847;
   DATA[775,30] := 1.731864;
   DATA[775,31] := 1.308569;
   DATA[775,32] := 0.7352687;
   DATA[775,33] := 0.3065048;
   DATA[775,34] := 2.0;
   DATA[775,35] := 250.9613;
   DATA[775,36] := 1.649953;
   DATA[775,37] := 189.759;
   DATA[775,38] := 0.000128152;
   DATA[775,39] := 1.0;
   DATA[776,0] := 2.537232;
   DATA[776,1] := 546.8694;
   DATA[776,2] := 2.0;
   DATA[776,3] := 1.0;
   DATA[776,4] := 262.1764;
   DATA[776,5] := 8.4429;
   DATA[776,6] := 318.8926;
   DATA[776,8] := 1.0;
   DATA[776,9] := 1.0;
   DATA[776,10] := 1.0;
   DATA[776,11] := 2.013573;
   DATA[776,13] := 1010.638;
   DATA[776,14] := 1.0;
   DATA[776,15] := 1.0;
   DATA[776,16] := 1.0;
   DATA[776,17] := 1.0;
   DATA[776,18] := 1.0;
   DATA[776,19] := 1.0;
   DATA[776,20] := 148.808;
   DATA[776,21] := 155.7293;
   DATA[776,22] := 1.717746;
   DATA[776,23] := 985.2089;
   DATA[776,24] := 2.0;
   DATA[776,25] := 2.0;
   DATA[776,26] := 7.878942;
   DATA[776,27] := 144.9628;
   DATA[776,28] := 263.1056;
   DATA[776,29] := 11.95847;
   DATA[776,30] := 1.731864;
   DATA[776,31] := 1.318432;
   DATA[776,32] := 0.7352687;
   DATA[776,33] := 0.3065048;
   DATA[776,34] := 2.0;
   DATA[776,35] := 250.9613;
   DATA[776,36] := 1.649953;
   DATA[776,37] := 189.759;
   DATA[776,38] := 0.000128152;
   DATA[776,39] := 1.0;
   DATA[777,0] := 2.542677;
   DATA[777,1] := 547.262;
   DATA[777,2] := 2.0;
   DATA[777,3] := 1.0;
   DATA[777,4] := 262.1764;
   DATA[777,5] := 8.444822;
   DATA[777,6] := 318.3799;
   DATA[777,8] := 1.0;
   DATA[777,9] := 1.0;
   DATA[777,10] := 1.0;
   DATA[777,11] := 2.013573;
   DATA[777,13] := 1010.839;
   DATA[777,14] := 1.0;
   DATA[777,15] := 1.0;
   DATA[777,16] := 1.0;
   DATA[777,17] := 1.0;
   DATA[777,18] := 1.0;
   DATA[777,19] := 1.0;
   DATA[777,20] := 148.808;
   DATA[777,21] := 155.7293;
   DATA[777,22] := 1.717361;
   DATA[777,23] := 984.5937;
   DATA[777,24] := 2.0;
   DATA[777,25] := 2.0;
   DATA[777,26] := 7.878942;
   DATA[777,27] := 144.9628;
   DATA[777,28] := 263.1056;
   DATA[777,29] := 11.95847;
   DATA[777,30] := 1.731864;
   DATA[777,31] := 1.321506;
   DATA[777,32] := 0.7352687;
   DATA[777,33] := 0.3065048;
   DATA[777,34] := 2.0;
   DATA[777,35] := 251.1055;
   DATA[777,36] := 1.649953;
   DATA[777,37] := 189.759;
   DATA[777,38] := 0.000128152;
   DATA[777,39] := 1.0;
   DATA[778,0] := 2.543958;
   DATA[778,1] := 547.6152;
   DATA[778,2] := 2.0;
   DATA[778,3] := 1.0;
   DATA[778,4] := 262.1764;
   DATA[778,5] := 8.449949;
   DATA[778,6] := 318.2774;
   DATA[778,8] := 1.0;
   DATA[778,9] := 1.0;
   DATA[778,10] := 1.0;
   DATA[778,11] := 2.013573;
   DATA[778,13] := 1010.758;
   DATA[778,14] := 1.0;
   DATA[778,15] := 1.0;
   DATA[778,16] := 1.0;
   DATA[778,17] := 1.0;
   DATA[778,18] := 1.0;
   DATA[778,19] := 1.0;
   DATA[778,20] := 148.808;
   DATA[778,21] := 155.7293;
   DATA[778,22] := 1.717233;
   DATA[778,23] := 984.4014;
   DATA[778,24] := 2.0;
   DATA[778,25] := 2.0;
   DATA[778,26] := 7.878942;
   DATA[778,27] := 144.9628;
   DATA[778,28] := 263.1056;
   DATA[778,29] := 11.95847;
   DATA[778,30] := 1.731864;
   DATA[778,31] := 1.31254;
   DATA[778,32] := 0.7352687;
   DATA[778,33] := 0.3065048;
   DATA[778,34] := 2.0;
   DATA[778,35] := 251.1055;
   DATA[778,36] := 1.649953;
   DATA[778,37] := 189.759;
   DATA[778,38] := 0.000128152;
   DATA[778,39] := 1.0;
   DATA[779,0] := 2.543958;
   DATA[779,1] := 547.4975;
   DATA[779,2] := 2.0;
   DATA[779,3] := 1.0;
   DATA[779,4] := 262.1764;
   DATA[779,5] := 8.452192;
   DATA[779,6] := 317.9954;
   DATA[779,8] := 1.0;
   DATA[779,9] := 1.0;
   DATA[779,10] := 1.0;
   DATA[779,11] := 2.013573;
   DATA[779,13] := 1010.758;
   DATA[779,14] := 1.0;
   DATA[779,15] := 1.0;
   DATA[779,16] := 1.0;
   DATA[779,17] := 1.0;
   DATA[779,18] := 1.0;
   DATA[779,19] := 1.0;
   DATA[779,20] := 148.808;
   DATA[779,21] := 155.7293;
   DATA[779,22] := 1.717233;
   DATA[779,23] := 983.7862;
   DATA[779,24] := 2.0;
   DATA[779,25] := 2.0;
   DATA[779,26] := 7.878942;
   DATA[779,27] := 144.9628;
   DATA[779,28] := 263.1056;
   DATA[779,29] := 11.95847;
   DATA[779,30] := 1.731864;
   DATA[779,31] := 1.304214;
   DATA[779,32] := 0.7352687;
   DATA[779,33] := 0.3065048;
   DATA[779,34] := 2.0;
   DATA[779,35] := 251.1055;
   DATA[779,36] := 1.649953;
   DATA[779,37] := 189.759;
   DATA[779,38] := 0.000128152;
   DATA[779,39] := 1.0;
   DATA[780,0] := 2.543958;
   DATA[780,1] := 547.4582;
   DATA[780,2] := 2.0;
   DATA[780,3] := 1.0;
   DATA[780,4] := 262.1764;
   DATA[780,5] := 8.452833;
   DATA[780,6] := 317.9185;
   DATA[780,8] := 1.0;
   DATA[780,9] := 1.0;
   DATA[780,10] := 1.0;
   DATA[780,11] := 2.013573;
   DATA[780,13] := 1010.638;
   DATA[780,14] := 1.0;
   DATA[780,15] := 1.0;
   DATA[780,16] := 1.0;
   DATA[780,17] := 1.0;
   DATA[780,18] := 1.0;
   DATA[780,19] := 1.0;
   DATA[780,20] := 148.808;
   DATA[780,21] := 155.7293;
   DATA[780,22] := 1.717233;
   DATA[780,23] := 983.5939;
   DATA[780,24] := 2.0;
   DATA[780,25] := 2.0;
   DATA[780,26] := 7.878942;
   DATA[780,27] := 144.9628;
   DATA[780,28] := 263.1056;
   DATA[780,29] := 11.95847;
   DATA[780,30] := 1.730582;
   DATA[780,31] := 1.297682;
   DATA[780,32] := 0.7352687;
   DATA[780,33] := 0.3065048;
   DATA[780,34] := 2.0;
   DATA[780,35] := 251.1055;
   DATA[780,36] := 1.649953;
   DATA[780,37] := 189.759;
   DATA[780,38] := 0.000128152;
   DATA[780,39] := 1.0;
   DATA[781,0] := 2.539474;
   DATA[781,1] := 547.4189;
   DATA[781,2] := 2.0;
   DATA[781,3] := 1.0;
   DATA[781,4] := 262.1764;
   DATA[781,5] := 8.452833;
   DATA[781,6] := 317.8672;
   DATA[781,8] := 1.0;
   DATA[781,9] := 1.0;
   DATA[781,10] := 1.0;
   DATA[781,11] := 2.013573;
   DATA[781,13] := 1010.758;
   DATA[781,14] := 1.0;
   DATA[781,15] := 1.0;
   DATA[781,16] := 1.0;
   DATA[781,17] := 1.0;
   DATA[781,18] := 1.0;
   DATA[781,19] := 1.0;
   DATA[781,20] := 148.808;
   DATA[781,21] := 155.7293;
   DATA[781,22] := 1.717233;
   DATA[781,23] := 983.0556;
   DATA[781,24] := 2.0;
   DATA[781,25] := 2.0;
   DATA[781,26] := 7.878942;
   DATA[781,27] := 144.9628;
   DATA[781,28] := 263.1056;
   DATA[781,29] := 11.95847;
   DATA[781,30] := 1.730582;
   DATA[781,31] := 1.291533;
   DATA[781,32] := 0.7352687;
   DATA[781,33] := 0.3065048;
   DATA[781,34] := 2.0;
   DATA[781,35] := 251.1055;
   DATA[781,36] := 1.69801;
   DATA[781,37] := 189.759;
   DATA[781,38] := 0.000128152;
   DATA[781,39] := 1.0;
   DATA[782,0] := 2.537873;
   DATA[782,1] := 547.9685;
   DATA[782,2] := 2.0;
   DATA[782,3] := 1.0;
   DATA[782,4] := 262.1764;
   DATA[782,5] := 8.456038;
   DATA[782,6] := 317.7903;
   DATA[782,8] := 1.0;
   DATA[782,9] := 1.0;
   DATA[782,10] := 1.0;
   DATA[782,11] := 2.042384;
   DATA[782,13] := 1010.438;
   DATA[782,14] := 1.0;
   DATA[782,15] := 1.0;
   DATA[782,16] := 1.0;
   DATA[782,17] := 1.0;
   DATA[782,18] := 1.0;
   DATA[782,19] := 1.0;
   DATA[782,20] := 148.808;
   DATA[782,21] := 155.7293;
   DATA[782,22] := 1.717233;
   DATA[782,23] := 982.4789;
   DATA[782,24] := 2.0;
   DATA[782,25] := 2.0;
   DATA[782,26] := 7.878942;
   DATA[782,27] := 144.9628;
   DATA[782,28] := 263.1056;
   DATA[782,29] := 11.95847;
   DATA[782,30] := 1.730582;
   DATA[782,31] := 1.291533;
   DATA[782,32] := 0.7352687;
   DATA[782,33] := 0.3065048;
   DATA[782,34] := 2.0;
   DATA[782,35] := 251.1055;
   DATA[782,36] := 1.69801;
   DATA[782,37] := 189.759;
   DATA[782,38] := 0.000128152;
   DATA[782,39] := 1.0;
   DATA[783,0] := 2.537873;
   DATA[783,1] := 548.9891;
   DATA[783,2] := 2.0;
   DATA[783,3] := 1.0;
   DATA[783,4] := 262.1764;
   DATA[783,5] := 8.456038;
   DATA[783,6] := 317.6109;
   DATA[783,8] := 1.0;
   DATA[783,9] := 1.0;
   DATA[783,10] := 1.0;
   DATA[783,11] := 2.042384;
   DATA[783,13] := 1010.518;
   DATA[783,14] := 1.0;
   DATA[783,15] := 1.0;
   DATA[783,16] := 1.0;
   DATA[783,17] := 1.0;
   DATA[783,18] := 1.0;
   DATA[783,19] := 1.0;
   DATA[783,20] := 148.808;
   DATA[783,21] := 155.7293;
   DATA[783,22] := 1.720309;
   DATA[783,23] := 982.4404;
   DATA[783,24] := 2.0;
   DATA[783,25] := 2.0;
   DATA[783,26] := 7.878942;
   DATA[783,27] := 144.9628;
   DATA[783,28] := 263.1056;
   DATA[783,29] := 11.95847;
   DATA[783,30] := 1.728788;
   DATA[783,31] := 1.295888;
   DATA[783,32] := 0.7352687;
   DATA[783,33] := 0.3065048;
   DATA[783,34] := 2.0;
   DATA[783,35] := 251.1055;
   DATA[783,36] := 1.69801;
   DATA[783,37] := 189.759;
   DATA[783,38] := 0.000128152;
   DATA[783,39] := 1.0;
   DATA[784,0] := 2.533709;
   DATA[784,1] := 549.7349;
   DATA[784,2] := 2.0;
   DATA[784,3] := 1.0;
   DATA[784,4] := 262.1764;
   DATA[784,5] := 8.456038;
   DATA[784,6] := 317.5083;
   DATA[784,8] := 1.0;
   DATA[784,9] := 1.0;
   DATA[784,10] := 1.0;
   DATA[784,11] := 2.042384;
   DATA[784,13] := 1010.678;
   DATA[784,14] := 1.0;
   DATA[784,15] := 1.0;
   DATA[784,16] := 1.0;
   DATA[784,17] := 1.0;
   DATA[784,18] := 1.0;
   DATA[784,19] := 1.0;
   DATA[784,20] := 148.808;
   DATA[784,21] := 155.7293;
   DATA[784,22] := 1.720309;
   DATA[784,23] := 982.2482;
   DATA[784,24] := 2.0;
   DATA[784,25] := 2.0;
   DATA[784,26] := 7.878942;
   DATA[784,27] := 144.9628;
   DATA[784,28] := 263.1056;
   DATA[784,29] := 11.95847;
   DATA[784,30] := 1.728788;
   DATA[784,31] := 1.291405;
   DATA[784,32] := 0.7352687;
   DATA[784,33] := 0.3065048;
   DATA[784,34] := 2.0;
   DATA[784,35] := 250.9613;
   DATA[784,36] := 1.69801;
   DATA[784,37] := 189.759;
   DATA[784,38] := 0.000128152;
   DATA[784,39] := 1.0;
   DATA[785,0] := 2.533709;
   DATA[785,1] := 549.6564;
   DATA[785,2] := 2.0;
   DATA[785,3] := 1.0;
   DATA[785,4] := 262.1764;
   DATA[785,5] := 8.45764;
   DATA[785,6] := 317.252;
   DATA[785,8] := 1.0;
   DATA[785,9] := 1.0;
   DATA[785,10] := 1.0;
   DATA[785,11] := 2.042384;
   DATA[785,13] := 1010.839;
   DATA[785,14] := 1.0;
   DATA[785,15] := 1.0;
   DATA[785,16] := 1.0;
   DATA[785,17] := 1.0;
   DATA[785,18] := 1.0;
   DATA[785,19] := 1.0;
   DATA[785,20] := 148.808;
   DATA[785,21] := 155.7293;
   DATA[785,22] := 1.720309;
   DATA[785,23] := 981.979;
   DATA[785,24] := 2.0;
   DATA[785,25] := 2.0;
   DATA[785,26] := 7.878942;
   DATA[785,27] := 144.9628;
   DATA[785,28] := 263.1056;
   DATA[785,29] := 11.95847;
   DATA[785,30] := 1.728788;
   DATA[785,31] := 1.282311;
   DATA[785,32] := 0.7352687;
   DATA[785,33] := 0.3065048;
   DATA[785,34] := 2.0;
   DATA[785,35] := 250.9453;
   DATA[785,36] := 1.69801;
   DATA[785,37] := 189.759;
   DATA[785,38] := 0.000128152;
   DATA[785,39] := 1.0;
   DATA[786,0] := 2.537232;
   DATA[786,1] := 550.4414;
   DATA[786,2] := 2.0;
   DATA[786,3] := 1.0;
   DATA[786,4] := 262.1764;
   DATA[786,5] := 8.461805;
   DATA[786,6] := 317.1751;
   DATA[786,8] := 1.0;
   DATA[786,9] := 1.0;
   DATA[786,10] := 1.0;
   DATA[786,11] := 2.042384;
   DATA[786,13] := 1010.678;
   DATA[786,14] := 1.0;
   DATA[786,15] := 1.0;
   DATA[786,16] := 1.0;
   DATA[786,17] := 1.0;
   DATA[786,18] := 1.0;
   DATA[786,19] := 1.0;
   DATA[786,20] := 148.808;
   DATA[786,21] := 155.5242;
   DATA[786,22] := 1.718002;
   DATA[786,23] := 981.7483;
   DATA[786,24] := 2.0;
   DATA[786,25] := 2.0;
   DATA[786,26] := 7.878942;
   DATA[786,27] := 144.9628;
   DATA[786,28] := 263.1056;
   DATA[786,29] := 11.95847;
   DATA[786,30] := 1.729428;
   DATA[786,31] := 1.286666;
   DATA[786,32] := 0.7352687;
   DATA[786,33] := 0.3065048;
   DATA[786,34] := 2.0;
   DATA[786,35] := 250.9453;
   DATA[786,36] := 1.746067;
   DATA[786,37] := 189.743;
   DATA[786,38] := 0.000128152;
   DATA[786,39] := 1.0;
   DATA[787,0] := 2.540115;
   DATA[787,1] := 551.1087;
   DATA[787,2] := 2.0;
   DATA[787,3] := 1.0;
   DATA[787,4] := 262.1764;
   DATA[787,5] := 8.461805;
   DATA[787,6] := 317.1751;
   DATA[787,8] := 1.0;
   DATA[787,9] := 1.0;
   DATA[787,10] := 1.0;
   DATA[787,11] := 2.042384;
   DATA[787,13] := 1010.638;
   DATA[787,14] := 1.0;
   DATA[787,15] := 1.0;
   DATA[787,16] := 1.0;
   DATA[787,17] := 1.0;
   DATA[787,18] := 1.0;
   DATA[787,19] := 1.0;
   DATA[787,20] := 148.808;
   DATA[787,21] := 155.5242;
   DATA[787,22] := 1.717874;
   DATA[787,23] := 981.3638;
   DATA[787,24] := 2.0;
   DATA[787,25] := 2.0;
   DATA[787,26] := 7.878942;
   DATA[787,27] := 144.9628;
   DATA[787,28] := 263.1056;
   DATA[787,29] := 11.95847;
   DATA[787,30] := 1.730197;
   DATA[787,31] := 1.280646;
   DATA[787,32] := 0.7352687;
   DATA[787,33] := 0.3065048;
   DATA[787,34] := 2.0;
   DATA[787,35] := 250.9453;
   DATA[787,36] := 1.746067;
   DATA[787,37] := 189.743;
   DATA[787,38] := 0.000128152;
   DATA[787,39] := 1.0;
   DATA[788,0] := 2.54652;
   DATA[788,1] := 551.619;
   DATA[788,2] := 2.0;
   DATA[788,3] := 1.0;
   DATA[788,4] := 262.1764;
   DATA[788,5] := 8.461805;
   DATA[788,6] := 317.1751;
   DATA[788,8] := 1.0;
   DATA[788,9] := 1.0;
   DATA[788,10] := 1.0;
   DATA[788,11] := 2.042384;
   DATA[788,13] := 1010.718;
   DATA[788,14] := 1.0;
   DATA[788,15] := 1.0;
   DATA[788,16] := 1.0;
   DATA[788,17] := 1.0;
   DATA[788,18] := 1.0;
   DATA[788,19] := 1.0;
   DATA[788,20] := 148.808;
   DATA[788,21] := 155.5242;
   DATA[788,22] := 1.717874;
   DATA[788,23] := 981.0946;
   DATA[788,24] := 2.0;
   DATA[788,25] := 2.0;
   DATA[788,26] := 7.878942;
   DATA[788,27] := 144.9628;
   DATA[788,28] := 263.1056;
   DATA[788,29] := 11.95847;
   DATA[788,30] := 1.730197;
   DATA[788,31] := 1.291533;
   DATA[788,32] := 0.7352687;
   DATA[788,33] := 0.3065048;
   DATA[788,34] := 2.0;
   DATA[788,35] := 250.9453;
   DATA[788,36] := 1.746067;
   DATA[788,37] := 189.743;
   DATA[788,38] := 0.000128152;
   DATA[788,39] := 1.0;
   DATA[789,0] := 2.547161;
   DATA[789,1] := 552.3648;
   DATA[789,2] := 2.0;
   DATA[789,3] := 1.0;
   DATA[789,4] := 262.1764;
   DATA[789,5] := 8.461805;
   DATA[789,6] := 317.1751;
   DATA[789,8] := 1.0;
   DATA[789,9] := 1.0;
   DATA[789,10] := 1.0;
   DATA[789,11] := 2.042384;
   DATA[789,13] := 1010.558;
   DATA[789,14] := 1.0;
   DATA[789,15] := 1.0;
   DATA[789,16] := 1.0;
   DATA[789,17] := 1.0;
   DATA[789,18] := 1.0;
   DATA[789,19] := 1.0;
   DATA[789,20] := 148.808;
   DATA[789,21] := 155.678;
   DATA[789,22] := 1.717874;
   DATA[789,23] := 980.9408;
   DATA[789,24] := 2.0;
   DATA[789,25] := 2.0;
   DATA[789,26] := 7.878942;
   DATA[789,27] := 145.1166;
   DATA[789,28] := 263.1056;
   DATA[789,29] := 11.95847;
   DATA[789,30] := 1.730197;
   DATA[789,31] := 1.291789;
   DATA[789,32] := 0.7352687;
   DATA[789,33] := 0.306761;
   DATA[789,34] := 2.0;
   DATA[789,35] := 250.9453;
   DATA[789,36] := 1.746067;
   DATA[789,37] := 189.6469;
   DATA[789,38] := 0.000128152;
   DATA[789,39] := 1.0;
   DATA[790,0] := 2.548762;
   DATA[790,1] := 553.1106;
   DATA[790,2] := 2.0;
   DATA[790,3] := 1.0;
   DATA[790,4] := 262.1764;
   DATA[790,5] := 8.461805;
   DATA[790,6] := 316.8675;
   DATA[790,8] := 1.0;
   DATA[790,9] := 1.0;
   DATA[790,10] := 1.0;
   DATA[790,11] := 2.042384;
   DATA[790,13] := 1011.039;
   DATA[790,14] := 1.0;
   DATA[790,15] := 1.0;
   DATA[790,16] := 1.0;
   DATA[790,17] := 1.0;
   DATA[790,18] := 1.0;
   DATA[790,19] := 1.0;
   DATA[790,20] := 148.808;
   DATA[790,21] := 155.7293;
   DATA[790,22] := 1.717874;
   DATA[790,23] := 980.364;
   DATA[790,24] := 2.0;
   DATA[790,25] := 2.0;
   DATA[790,26] := 7.878942;
   DATA[790,27] := 145.1423;
   DATA[790,28] := 263.1056;
   DATA[790,29] := 11.95847;
   DATA[790,30] := 1.728531;
   DATA[790,31] := 1.281798;
   DATA[790,32] := 0.7352687;
   DATA[790,33] := 0.3069532;
   DATA[790,34] := 2.0;
   DATA[790,35] := 250.9453;
   DATA[790,36] := 1.746067;
   DATA[790,37] := 189.6469;
   DATA[790,38] := 0.000128152;
   DATA[790,39] := 1.0;
   DATA[791,0] := 2.550043;
   DATA[791,1] := 554.0527;
   DATA[791,2] := 2.0;
   DATA[791,3] := 1.0;
   DATA[791,4] := 262.1764;
   DATA[791,5] := 8.461805;
   DATA[791,6] := 316.8675;
   DATA[791,8] := 1.0;
   DATA[791,9] := 1.0;
   DATA[791,10] := 1.0;
   DATA[791,11] := 2.042384;
   DATA[791,13] := 1011.119;
   DATA[791,14] := 1.0;
   DATA[791,15] := 1.0;
   DATA[791,16] := 1.0;
   DATA[791,17] := 1.0;
   DATA[791,18] := 1.0;
   DATA[791,19] := 1.0;
   DATA[791,20] := 148.808;
   DATA[791,21] := 155.7293;
   DATA[791,22] := 1.717874;
   DATA[791,23] := 979.6719;
   DATA[791,24] := 2.0;
   DATA[791,25] := 2.0;
   DATA[791,26] := 7.878942;
   DATA[791,27] := 145.1423;
   DATA[791,28] := 263.1056;
   DATA[791,29] := 11.95847;
   DATA[791,30] := 1.728531;
   DATA[791,31] := 1.274625;
   DATA[791,32] := 0.7352687;
   DATA[791,33] := 0.3069532;
   DATA[791,34] := 2.0;
   DATA[791,35] := 250.9453;
   DATA[791,36] := 1.746067;
   DATA[791,37] := 189.6469;
   DATA[791,38] := 0.000128152;
   DATA[791,39] := 1.0;
   DATA[792,0] := 2.551965;
   DATA[792,1] := 554.6807;
   DATA[792,2] := 2.0;
   DATA[792,3] := 1.0;
   DATA[792,4] := 262.1764;
   DATA[792,5] := 8.46533;
   DATA[792,6] := 316.8675;
   DATA[792,8] := 1.0;
   DATA[792,9] := 1.0;
   DATA[792,10] := 1.0;
   DATA[792,11] := 2.042384;
   DATA[792,13] := 1011.159;
   DATA[792,14] := 1.0;
   DATA[792,15] := 1.0;
   DATA[792,16] := 1.0;
   DATA[792,17] := 1.0;
   DATA[792,18] := 1.0;
   DATA[792,19] := 1.0;
   DATA[792,20] := 148.808;
   DATA[792,21] := 155.7293;
   DATA[792,22] := 1.717874;
   DATA[792,23] := 979.4796;
   DATA[792,24] := 2.0;
   DATA[792,25] := 2.0;
   DATA[792,26] := 7.878942;
   DATA[792,27] := 145.1423;
   DATA[792,28] := 263.0415;
   DATA[792,29] := 11.95847;
   DATA[792,30] := 1.728531;
   DATA[792,31] := 1.263866;
   DATA[792,32] := 0.7352687;
   DATA[792,33] := 0.3069532;
   DATA[792,34] := 2.0;
   DATA[792,35] := 250.9453;
   DATA[792,36] := 1.746067;
   DATA[792,37] := 189.6469;
   DATA[792,38] := 0.000128152;
   DATA[792,39] := 1.0;
   DATA[793,0] := 2.552926;
   DATA[793,1] := 555.4265;
   DATA[793,2] := 2.0;
   DATA[793,3] := 1.0;
   DATA[793,4] := 262.1764;
   DATA[793,5] := 8.46533;
   DATA[793,6] := 316.7137;
   DATA[793,8] := 1.0;
   DATA[793,9] := 1.0;
   DATA[793,10] := 1.0;
   DATA[793,11] := 2.042384;
   DATA[793,13] := 1010.839;
   DATA[793,14] := 1.0;
   DATA[793,15] := 1.0;
   DATA[793,16] := 1.0;
   DATA[793,17] := 1.0;
   DATA[793,18] := 1.0;
   DATA[793,19] := 1.0;
   DATA[793,20] := 148.808;
   DATA[793,21] := 155.7293;
   DATA[793,22] := 1.717874;
   DATA[793,23] := 978.9797;
   DATA[793,24] := 2.0;
   DATA[793,25] := 2.0;
   DATA[793,26] := 7.878942;
   DATA[793,27] := 145.1423;
   DATA[793,28] := 263.0415;
   DATA[793,29] := 11.95847;
   DATA[793,30] := 1.728531;
   DATA[793,31] := 1.262713;
   DATA[793,32] := 0.7352687;
   DATA[793,33] := 0.3075937;
   DATA[793,34] := 2.0;
   DATA[793,35] := 250.8171;
   DATA[793,36] := 1.746067;
   DATA[793,37] := 189.6469;
   DATA[793,38] := 0.000128152;
   DATA[793,39] := 1.0;
   DATA[794,0] := 2.552926;
   DATA[794,1] := 555.819;
   DATA[794,2] := 2.0;
   DATA[794,3] := 1.0;
   DATA[794,4] := 262.1764;
   DATA[794,5] := 8.46533;
   DATA[794,6] := 316.5086;
   DATA[794,8] := 1.0;
   DATA[794,9] := 1.0;
   DATA[794,10] := 1.0;
   DATA[794,11] := 2.042384;
   DATA[794,13] := 1011.079;
   DATA[794,14] := 1.0;
   DATA[794,15] := 1.0;
   DATA[794,16] := 1.0;
   DATA[794,17] := 1.0;
   DATA[794,18] := 1.0;
   DATA[794,19] := 1.0;
   DATA[794,20] := 148.808;
   DATA[794,21] := 155.7293;
   DATA[794,22] := 1.717874;
   DATA[794,23] := 978.9797;
   DATA[794,24] := 2.0;
   DATA[794,25] := 2.0;
   DATA[794,26] := 7.878942;
   DATA[794,27] := 145.1166;
   DATA[794,28] := 263.0415;
   DATA[794,29] := 11.95847;
   DATA[794,30] := 1.726352;
   DATA[794,31] := 1.278084;
   DATA[794,32] := 0.7352687;
   DATA[794,33] := 0.3077859;
   DATA[794,34] := 2.0;
   DATA[794,35] := 250.8171;
   DATA[794,36] := 1.746067;
   DATA[794,37] := 189.6469;
   DATA[794,38] := 0.000128152;
   DATA[794,39] := 1.0;
   DATA[795,0] := 2.552926;
   DATA[795,1] := 556.1723;
   DATA[795,2] := 2.0;
   DATA[795,3] := 1.0;
   DATA[795,4] := 262.1764;
   DATA[795,5] := 8.46533;
   DATA[795,6] := 316.5086;
   DATA[795,8] := 1.0;
   DATA[795,9] := 1.0;
   DATA[795,10] := 1.0;
   DATA[795,11] := 2.042384;
   DATA[795,13] := 1010.518;
   DATA[795,14] := 1.0;
   DATA[795,15] := 1.0;
   DATA[795,16] := 1.0;
   DATA[795,17] := 1.0;
   DATA[795,18] := 1.0;
   DATA[795,19] := 1.0;
   DATA[795,20] := 148.808;
   DATA[795,21] := 155.7293;
   DATA[795,22] := 1.717874;
   DATA[795,23] := 978.8259;
   DATA[795,24] := 2.0;
   DATA[795,25] := 2.0;
   DATA[795,26] := 7.878942;
   DATA[795,27] := 144.9116;
   DATA[795,28] := 263.0415;
   DATA[795,29] := 11.95847;
   DATA[795,30] := 1.726352;
   DATA[795,31] := 1.289356;
   DATA[795,32] := 0.7352687;
   DATA[795,33] := 0.306761;
   DATA[795,34] := 2.0;
   DATA[795,35] := 250.8171;
   DATA[795,36] := 1.69801;
   DATA[795,37] := 189.6469;
   DATA[795,38] := 0.000128152;
   DATA[795,39] := 1.0;
   DATA[796,0] := 2.548442;
   DATA[796,1] := 556.5649;
   DATA[796,2] := 2.0;
   DATA[796,3] := 1.0;
   DATA[796,4] := 262.1764;
   DATA[796,5] := 8.46533;
   DATA[796,6] := 316.4573;
   DATA[796,8] := 1.0;
   DATA[796,9] := 1.0;
   DATA[796,10] := 1.0;
   DATA[796,11] := 2.042384;
   DATA[796,13] := 1010.959;
   DATA[796,14] := 1.0;
   DATA[796,15] := 1.0;
   DATA[796,16] := 1.0;
   DATA[796,17] := 1.0;
   DATA[796,18] := 1.0;
   DATA[796,19] := 1.0;
   DATA[796,20] := 148.808;
   DATA[796,21] := 155.7293;
   DATA[796,22] := 1.717874;
   DATA[796,23] := 978.9028;
   DATA[796,24] := 2.0;
   DATA[796,25] := 2.0;
   DATA[796,26] := 7.878942;
   DATA[796,27] := 144.9116;
   DATA[796,28] := 263.0415;
   DATA[796,29] := 11.95847;
   DATA[796,30] := 1.726352;
   DATA[796,31] := 1.300115;
   DATA[796,32] := 0.7352687;
   DATA[796,33] := 0.3066329;
   DATA[796,34] := 2.0;
   DATA[796,35] := 250.8171;
   DATA[796,36] := 1.69801;
   DATA[796,37] := 189.6469;
   DATA[796,38] := 0.000128152;
   DATA[796,39] := 1.0;
   DATA[797,0] := 2.548442;
   DATA[797,1] := 556.9574;
   DATA[797,2] := 2.0;
   DATA[797,3] := 1.0;
   DATA[797,4] := 262.1764;
   DATA[797,5] := 8.46533;
   DATA[797,6] := 316.2522;
   DATA[797,8] := 1.0;
   DATA[797,9] := 1.0;
   DATA[797,10] := 1.0;
   DATA[797,11] := 2.042384;
   DATA[797,13] := 1010.959;
   DATA[797,14] := 1.0;
   DATA[797,15] := 1.0;
   DATA[797,16] := 1.0;
   DATA[797,17] := 1.0;
   DATA[797,18] := 1.0;
   DATA[797,19] := 1.0;
   DATA[797,20] := 148.808;
   DATA[797,21] := 155.7293;
   DATA[797,22] := 1.717874;
   DATA[797,23] := 978.5183;
   DATA[797,24] := 2.0;
   DATA[797,25] := 2.0;
   DATA[797,26] := 7.878942;
   DATA[797,27] := 144.9116;
   DATA[797,28] := 263.0415;
   DATA[797,29] := 11.95847;
   DATA[797,30] := 1.726352;
   DATA[797,31] := 1.30114;
   DATA[797,32] := 0.7352687;
   DATA[797,33] := 0.3066329;
   DATA[797,34] := 2.0;
   DATA[797,35] := 250.8171;
   DATA[797,36] := 1.69801;
   DATA[797,37] := 189.5828;
   DATA[797,38] := 0.000128152;
   DATA[797,39] := 1.0;
   DATA[798,0] := 2.548442;
   DATA[798,1] := 557.2322;
   DATA[798,2] := 2.0;
   DATA[798,3] := 1.0;
   DATA[798,4] := 262.1764;
   DATA[798,5] := 8.46533;
   DATA[798,6] := 316.2522;
   DATA[798,8] := 1.0;
   DATA[798,9] := 1.0;
   DATA[798,10] := 1.0;
   DATA[798,11] := 2.032781;
   DATA[798,13] := 1011.079;
   DATA[798,14] := 1.0;
   DATA[798,15] := 1.0;
   DATA[798,16] := 1.0;
   DATA[798,17] := 1.0;
   DATA[798,18] := 1.0;
   DATA[798,19] := 1.0;
   DATA[798,20] := 148.808;
   DATA[798,21] := 155.7293;
   DATA[798,22] := 1.717874;
   DATA[798,23] := 978.5183;
   DATA[798,24] := 2.0;
   DATA[798,25] := 2.0;
   DATA[798,26] := 7.878942;
   DATA[798,27] := 144.9116;
   DATA[798,28] := 263.0415;
   DATA[798,29] := 11.95847;
   DATA[798,30] := 1.726352;
   DATA[798,31] := 1.296657;
   DATA[798,32] := 0.7352687;
   DATA[798,33] := 0.3083624;
   DATA[798,34] := 2.0;
   DATA[798,35] := 250.8171;
   DATA[798,36] := 1.69801;
   DATA[798,37] := 189.4867;
   DATA[798,38] := 0.000128152;
   DATA[798,39] := 1.0;
   DATA[799,0] := 2.550684;
   DATA[799,1] := 557.6247;
   DATA[799,2] := 2.0;
   DATA[799,3] := 1.0;
   DATA[799,4] := 262.1764;
   DATA[799,5] := 8.46533;
   DATA[799,6] := 316.2522;
   DATA[799,8] := 1.0;
   DATA[799,9] := 1.0;
   DATA[799,10] := 1.0;
   DATA[799,11] := 2.032781;
   DATA[799,13] := 1010.879;
   DATA[799,14] := 1.0;
   DATA[799,15] := 1.0;
   DATA[799,16] := 1.0;
   DATA[799,17] := 1.0;
   DATA[799,18] := 1.0;
   DATA[799,19] := 1.0;
   DATA[799,20] := 148.808;
   DATA[799,21] := 155.7293;
   DATA[799,22] := 1.717874;
   DATA[799,23] := 977.8646;
   DATA[799,24] := 2.0;
   DATA[799,25] := 2.0;
   DATA[799,26] := 7.878942;
   DATA[799,27] := 144.9116;
   DATA[799,28] := 263.0415;
   DATA[799,29] := 11.95847;
   DATA[799,30] := 1.726352;
   DATA[799,31] := 1.301396;
   DATA[799,32] := 0.7352687;
   DATA[799,33] := 0.3083624;
   DATA[799,34] := 2.0;
   DATA[799,35] := 250.6569;
   DATA[799,36] := 1.69801;
   DATA[799,37] := 189.4867;
   DATA[799,38] := 0.000128152;
   DATA[799,39] := 1.0;
   DATA[800,0] := 2.553246;
   DATA[800,1] := 558.3705;
   DATA[800,2] := 2.0;
   DATA[800,3] := 1.0;
   DATA[800,4] := 262.1764;
   DATA[800,5] := 8.46533;
   DATA[800,6] := 316.2522;
   DATA[800,8] := 1.0;
   DATA[800,9] := 1.0;
   DATA[800,10] := 1.0;
   DATA[800,11] := 2.032781;
   DATA[800,13] := 1011.359;
   DATA[800,14] := 1.0;
   DATA[800,15] := 1.0;
   DATA[800,16] := 1.0;
   DATA[800,17] := 1.0;
   DATA[800,18] := 1.0;
   DATA[800,19] := 1.0;
   DATA[800,20] := 148.808;
   DATA[800,21] := 155.7293;
   DATA[800,22] := 1.717874;
   DATA[800,23] := 977.4417;
   DATA[800,24] := 2.0;
   DATA[800,25] := 2.0;
   DATA[800,26] := 7.878942;
   DATA[800,27] := 144.9116;
   DATA[800,28] := 263.0415;
   DATA[800,29] := 11.95847;
   DATA[800,30] := 1.726352;
   DATA[800,31] := 1.301396;
   DATA[800,32] := 0.7352687;
   DATA[800,33] := 0.3083624;
   DATA[800,34] := 2.0;
   DATA[800,35] := 250.6569;
   DATA[800,36] := 1.69801;
   DATA[800,37] := 189.4867;
   DATA[800,38] := 0.000128152;
   DATA[800,39] := 1.0;
   DATA[801,0] := 2.553246;
   DATA[801,1] := 559.3911;
   DATA[801,2] := 2.0;
   DATA[801,3] := 1.0;
   DATA[801,4] := 262.1764;
   DATA[801,5] := 8.46533;
   DATA[801,6] := 316.0984;
   DATA[801,8] := 1.0;
   DATA[801,9] := 1.0;
   DATA[801,10] := 1.0;
   DATA[801,11] := 2.032781;
   DATA[801,13] := 1011.119;
   DATA[801,14] := 1.0;
   DATA[801,15] := 1.0;
   DATA[801,16] := 1.0;
   DATA[801,17] := 1.0;
   DATA[801,18] := 1.0;
   DATA[801,19] := 1.0;
   DATA[801,20] := 148.808;
   DATA[801,21] := 155.7293;
   DATA[801,22] := 1.717874;
   DATA[801,23] := 976.9034;
   DATA[801,24] := 2.0;
   DATA[801,25] := 2.0;
   DATA[801,26] := 7.878942;
   DATA[801,27] := 144.9116;
   DATA[801,28] := 263.0415;
   DATA[801,29] := 11.95847;
   DATA[801,30] := 1.726352;
   DATA[801,31] := 1.302037;
   DATA[801,32] := 0.7352687;
   DATA[801,33] := 0.3083624;
   DATA[801,34] := 2.0;
   DATA[801,35] := 250.6569;
   DATA[801,36] := 1.69801;
   DATA[801,37] := 189.4867;
   DATA[801,38] := 0.000128152;
   DATA[801,39] := 1.0;
   DATA[802,0] := 2.553246;
   DATA[802,1] := 560.0191;
   DATA[802,2] := 2.0;
   DATA[802,3] := 1.0;
   DATA[802,4] := 262.1764;
   DATA[802,5] := 8.46533;
   DATA[802,6] := 316.0984;
   DATA[802,8] := 1.0;
   DATA[802,9] := 1.0;
   DATA[802,10] := 1.0;
   DATA[802,11] := 2.032781;
   DATA[802,13] := 1011.159;
   DATA[802,14] := 1.0;
   DATA[802,15] := 1.0;
   DATA[802,16] := 1.0;
   DATA[802,17] := 1.0;
   DATA[802,18] := 1.0;
   DATA[802,19] := 1.0;
   DATA[802,20] := 148.808;
   DATA[802,21] := 155.7293;
   DATA[802,22] := 1.717874;
   DATA[802,23] := 976.5573;
   DATA[802,24] := 2.0;
   DATA[802,25] := 2.0;
   DATA[802,26] := 7.878942;
   DATA[802,27] := 144.9116;
   DATA[802,28] := 263.0415;
   DATA[802,29] := 11.95847;
   DATA[802,30] := 1.72725;
   DATA[802,31] := 1.30178;
   DATA[802,32] := 0.7352687;
   DATA[802,33] := 0.3083624;
   DATA[802,34] := 2.0;
   DATA[802,35] := 250.6569;
   DATA[802,36] := 1.69801;
   DATA[802,37] := 189.4867;
   DATA[802,38] := 0.000128152;
   DATA[802,39] := 1.0;
   DATA[803,0] := 2.549082;
   DATA[803,1] := 561.0004;
   DATA[803,2] := 2.0;
   DATA[803,3] := 1.0;
   DATA[803,4] := 262.5288;
   DATA[803,5] := 8.46533;
   DATA[803,6] := 316.0984;
   DATA[803,8] := 1.0;
   DATA[803,9] := 1.0;
   DATA[803,10] := 1.0;
   DATA[803,11] := 2.032781;
   DATA[803,13] := 1010.879;
   DATA[803,14] := 1.0;
   DATA[803,15] := 1.0;
   DATA[803,16] := 1.0;
   DATA[803,17] := 1.0;
   DATA[803,18] := 1.0;
   DATA[803,19] := 1.0;
   DATA[803,20] := 148.808;
   DATA[803,21] := 155.7293;
   DATA[803,22] := 1.717874;
   DATA[803,23] := 976.3651;
   DATA[803,24] := 2.0;
   DATA[803,25] := 2.0;
   DATA[803,26] := 7.878942;
   DATA[803,27] := 145.0141;
   DATA[803,28] := 263.0415;
   DATA[803,29] := 11.95847;
   DATA[803,30] := 1.72725;
   DATA[803,31] := 1.284104;
   DATA[803,32] := 0.7352687;
   DATA[803,33] := 0.3083624;
   DATA[803,34] := 2.0;
   DATA[803,35] := 250.6569;
   DATA[803,36] := 1.778105;
   DATA[803,37] := 189.4867;
   DATA[803,38] := 0.000128152;
   DATA[803,39] := 1.0;
   DATA[804,0] := 2.54652;
   DATA[804,1] := 561.9033;
   DATA[804,2] := 2.0;
   DATA[804,3] := 1.0;
   DATA[804,4] := 262.5288;
   DATA[804,5] := 8.46533;
   DATA[804,6] := 315.9959;
   DATA[804,8] := 1.0;
   DATA[804,9] := 1.0;
   DATA[804,10] := 1.0;
   DATA[804,11] := 2.032781;
   DATA[804,13] := 1010.879;
   DATA[804,14] := 1.0;
   DATA[804,15] := 1.0;
   DATA[804,16] := 1.0;
   DATA[804,17] := 1.0;
   DATA[804,18] := 1.0;
   DATA[804,19] := 1.0;
   DATA[804,20] := 148.808;
   DATA[804,21] := 155.7293;
   DATA[804,22] := 1.717874;
   DATA[804,23] := 976.1728;
   DATA[804,24] := 2.0;
   DATA[804,25] := 2.0;
   DATA[804,26] := 7.878942;
   DATA[804,27] := 145.0141;
   DATA[804,28] := 263.0415;
   DATA[804,29] := 12.03538;
   DATA[804,30] := 1.72725;
   DATA[804,31] := 1.267709;
   DATA[804,32] := 0.7352687;
   DATA[804,33] := 0.3080421;
   DATA[804,34] := 2.0;
   DATA[804,35] := 250.737;
   DATA[804,36] := 1.778105;
   DATA[804,37] := 189.4867;
   DATA[804,38] := 0.000128152;
   DATA[804,39] := 1.0;
   DATA[805,0] := 2.54652;
   DATA[805,1] := 562.8845;
   DATA[805,2] := 2.0;
   DATA[805,3] := 1.0;
   DATA[805,4] := 262.5288;
   DATA[805,5] := 8.46533;
   DATA[805,6] := 315.8677;
   DATA[805,8] := 1.0;
   DATA[805,9] := 1.0;
   DATA[805,10] := 1.0;
   DATA[805,11] := 2.032781;
   DATA[805,13] := 1011.079;
   DATA[805,14] := 1.0;
   DATA[805,15] := 1.0;
   DATA[805,16] := 1.0;
   DATA[805,17] := 1.0;
   DATA[805,18] := 1.0;
   DATA[805,19] := 1.0;
   DATA[805,20] := 148.808;
   DATA[805,21] := 155.7293;
   DATA[805,22] := 1.717874;
   DATA[805,23] := 975.9421;
   DATA[805,24] := 2.0;
   DATA[805,25] := 2.0;
   DATA[805,26] := 7.878942;
   DATA[805,27] := 145.0141;
   DATA[805,28] := 263.0415;
   DATA[805,29] := 12.22763;
   DATA[805,30] := 1.72725;
   DATA[805,31] := 1.261688;
   DATA[805,32] := 0.7352687;
   DATA[805,33] := 0.3069532;
   DATA[805,34] := 2.0;
   DATA[805,35] := 250.785;
   DATA[805,36] := 1.778105;
   DATA[805,37] := 189.4867;
   DATA[805,38] := 0.000128152;
   DATA[805,39] := 1.0;
   DATA[806,0] := 2.54652;
   DATA[806,1] := 563.9052;
   DATA[806,2] := 2.0;
   DATA[806,3] := 1.0;
   DATA[806,4] := 262.2404;
   DATA[806,5] := 8.46533;
   DATA[806,6] := 315.8677;
   DATA[806,8] := 1.0;
   DATA[806,9] := 1.0;
   DATA[806,10] := 1.0;
   DATA[806,11] := 2.032781;
   DATA[806,13] := 1011.119;
   DATA[806,14] := 1.0;
   DATA[806,15] := 1.0;
   DATA[806,16] := 1.0;
   DATA[806,17] := 1.0;
   DATA[806,18] := 1.0;
   DATA[806,19] := 1.0;
   DATA[806,20] := 148.808;
   DATA[806,21] := 155.7293;
   DATA[806,22] := 1.717874;
   DATA[806,23] := 975.596;
   DATA[806,24] := 2.0;
   DATA[806,25] := 2.0;
   DATA[806,26] := 7.878942;
   DATA[806,27] := 145.0141;
   DATA[806,28] := 263.0415;
   DATA[806,29] := 12.22763;
   DATA[806,30] := 1.72725;
   DATA[806,31] := 1.255284;
   DATA[806,32] := 0.7352687;
   DATA[806,33] := 0.3069532;
   DATA[806,34] := 2.0;
   DATA[806,35] := 250.785;
   DATA[806,36] := 1.778105;
   DATA[806,37] := 189.4867;
   DATA[806,38] := 0.000128152;
   DATA[806,39] := 1.0;
   DATA[807,0] := 2.540115;
   DATA[807,1] := 564.8079;
   DATA[807,2] := 2.0;
   DATA[807,3] := 1.0;
   DATA[807,4] := 262.2404;
   DATA[807,5] := 8.46533;
   DATA[807,6] := 315.7396;
   DATA[807,8] := 1.0;
   DATA[807,9] := 1.0;
   DATA[807,10] := 1.0;
   DATA[807,11] := 2.032781;
   DATA[807,13] := 1011.359;
   DATA[807,14] := 1.0;
   DATA[807,15] := 1.0;
   DATA[807,16] := 1.0;
   DATA[807,17] := 1.0;
   DATA[807,18] := 1.0;
   DATA[807,19] := 1.0;
   DATA[807,20] := 148.808;
   DATA[807,21] := 155.7293;
   DATA[807,22] := 1.717874;
   DATA[807,23] := 975.0192;
   DATA[807,24] := 2.0;
   DATA[807,25] := 2.0;
   DATA[807,26] := 7.878942;
   DATA[807,27] := 145.0141;
   DATA[807,28] := 263.0415;
   DATA[807,29] := 12.22763;
   DATA[807,30] := 1.72725;
   DATA[807,31] := 1.254771;
   DATA[807,32] := 0.7352687;
   DATA[807,33] := 0.3081703;
   DATA[807,34] := 2.0;
   DATA[807,35] := 250.785;
   DATA[807,36] := 1.778105;
   DATA[807,37] := 189.4867;
   DATA[807,38] := 0.000128152;
   DATA[807,39] := 1.0;
   DATA[808,0] := 2.540115;
   DATA[808,1] := 565.2004;
   DATA[808,2] := 2.0;
   DATA[808,3] := 1.0;
   DATA[808,4] := 262.2404;
   DATA[808,5] := 8.46533;
   DATA[808,6] := 315.5858;
   DATA[808,8] := 1.0;
   DATA[808,9] := 1.0;
   DATA[808,10] := 1.0;
   DATA[808,11] := 2.032781;
   DATA[808,13] := 1010.919;
   DATA[808,14] := 1.0;
   DATA[808,15] := 1.0;
   DATA[808,16] := 1.0;
   DATA[808,17] := 1.0;
   DATA[808,18] := 1.0;
   DATA[808,19] := 1.0;
   DATA[808,20] := 148.808;
   DATA[808,21] := 155.7293;
   DATA[808,22] := 1.717874;
   DATA[808,23] := 974.6732;
   DATA[808,24] := 2.0;
   DATA[808,25] := 2.0;
   DATA[808,26] := 7.878942;
   DATA[808,27] := 145.0141;
   DATA[808,28] := 263.0415;
   DATA[808,29] := 12.22763;
   DATA[808,30] := 1.729172;
   DATA[808,31] := 1.270142;
   DATA[808,32] := 0.7352687;
   DATA[808,33] := 0.3081703;
   DATA[808,34] := 2.0;
   DATA[808,35] := 250.6729;
   DATA[808,36] := 1.649953;
   DATA[808,37] := 189.4867;
   DATA[808,38] := 0.000128152;
   DATA[808,39] := 1.0;
   DATA[809,0] := 2.551645;
   DATA[809,1] := 565.3967;
   DATA[809,2] := 2.0;
   DATA[809,3] := 1.0;
   DATA[809,4] := 262.2404;
   DATA[809,5] := 8.46533;
   DATA[809,6] := 315.5858;
   DATA[809,8] := 1.0;
   DATA[809,9] := 1.0;
   DATA[809,10] := 1.0;
   DATA[809,11] := 2.032781;
   DATA[809,13] := 1010.959;
   DATA[809,14] := 1.0;
   DATA[809,15] := 1.0;
   DATA[809,16] := 1.0;
   DATA[809,17] := 1.0;
   DATA[809,18] := 1.0;
   DATA[809,19] := 1.0;
   DATA[809,20] := 148.808;
   DATA[809,21] := 155.7293;
   DATA[809,22] := 1.717874;
   DATA[809,23] := 974.6347;
   DATA[809,24] := 2.0;
   DATA[809,25] := 2.0;
   DATA[809,26] := 7.878942;
   DATA[809,27] := 144.7578;
   DATA[809,28] := 263.0415;
   DATA[809,29] := 12.22763;
   DATA[809,30] := 1.729172;
   DATA[809,31] := 1.272576;
   DATA[809,32] := 0.7352687;
   DATA[809,33] := 0.3083624;
   DATA[809,34] := 2.0;
   DATA[809,35] := 250.5608;
   DATA[809,36] := 1.649953;
   DATA[809,37] := 189.3425;
   DATA[809,38] := 0.000128152;
   DATA[809,39] := 1.0;
   DATA[810,0] := 2.553886;
   DATA[810,1] := 565.5145;
   DATA[810,2] := 2.0;
   DATA[810,3] := 1.0;
   DATA[810,4] := 262.2404;
   DATA[810,5] := 8.46533;
   DATA[810,6] := 315.5601;
   DATA[810,8] := 1.0;
   DATA[810,9] := 1.0;
   DATA[810,10] := 1.0;
   DATA[810,11] := 2.032781;
   DATA[810,13] := 1011.039;
   DATA[810,14] := 1.0;
   DATA[810,15] := 1.0;
   DATA[810,16] := 1.0;
   DATA[810,17] := 1.0;
   DATA[810,18] := 1.0;
   DATA[810,19] := 1.0;
   DATA[810,20] := 148.808;
   DATA[810,21] := 155.7293;
   DATA[810,22] := 1.716849;
   DATA[810,23] := 974.1733;
   DATA[810,24] := 2.0;
   DATA[810,25] := 2.0;
   DATA[810,26] := 7.878942;
   DATA[810,27] := 144.7578;
   DATA[810,28] := 263.0415;
   DATA[810,29] := 12.22763;
   DATA[810,30] := 1.7293;
   DATA[810,31] := 1.272576;
   DATA[810,32] := 0.7352687;
   DATA[810,33] := 0.3072735;
   DATA[810,34] := 2.0;
   DATA[810,35] := 250.5608;
   DATA[810,36] := 1.649953;
   DATA[810,37] := 189.3425;
   DATA[810,38] := 0.000128152;
   DATA[810,39] := 1.0;
   DATA[811,0] := 2.554527;
   DATA[811,1] := 565.279;
   DATA[811,2] := 2.0;
   DATA[811,3] := 1.0;
   DATA[811,4] := 262.2404;
   DATA[811,5] := 8.46533;
   DATA[811,6] := 315.5601;
   DATA[811,8] := 1.0;
   DATA[811,9] := 1.0;
   DATA[811,10] := 1.0;
   DATA[811,11] := 2.032781;
   DATA[811,13] := 1010.718;
   DATA[811,14] := 1.0;
   DATA[811,15] := 1.0;
   DATA[811,16] := 1.0;
   DATA[811,17] := 1.0;
   DATA[811,18] := 1.0;
   DATA[811,19] := 1.0;
   DATA[811,20] := 148.808;
   DATA[811,21] := 155.7293;
   DATA[811,22] := 1.71608;
   DATA[811,23] := 973.7888;
   DATA[811,24] := 2.0;
   DATA[811,25] := 2.0;
   DATA[811,26] := 7.878942;
   DATA[811,27] := 144.7578;
   DATA[811,28] := 263.0415;
   DATA[811,29] := 11.84312;
   DATA[811,30] := 1.7293;
   DATA[811,31] := 1.272192;
   DATA[811,32] := 0.7352687;
   DATA[811,33] := 0.3068251;
   DATA[811,34] := 2.0;
   DATA[811,35] := 250.5608;
   DATA[811,36] := 1.649953;
   DATA[811,37] := 189.3425;
   DATA[811,38] := 0.000128152;
   DATA[811,39] := 1.0;
   DATA[812,0] := 2.554527;
   DATA[812,1] := 565.2397;
   DATA[812,2] := 2.0;
   DATA[812,3] := 1.0;
   DATA[812,4] := 262.2404;
   DATA[812,5] := 8.46533;
   DATA[812,6] := 315.5601;
   DATA[812,8] := 1.0;
   DATA[812,9] := 1.0;
   DATA[812,10] := 1.0;
   DATA[812,11] := 2.032781;
   DATA[812,13] := 1010.278;
   DATA[812,14] := 1.0;
   DATA[812,15] := 1.0;
   DATA[812,16] := 1.0;
   DATA[812,17] := 1.0;
   DATA[812,18] := 1.0;
   DATA[812,19] := 1.0;
   DATA[812,20] := 148.808;
   DATA[812,21] := 155.7293;
   DATA[812,22] := 1.715567;
   DATA[812,23] := 973.2889;
   DATA[812,24] := 2.0;
   DATA[812,25] := 2.0;
   DATA[812,26] := 7.878942;
   DATA[812,27] := 144.7578;
   DATA[812,28] := 263.0415;
   DATA[812,29] := 11.84312;
   DATA[812,30] := 1.7293;
   DATA[812,31] := 1.272576;
   DATA[812,32] := 0.7352687;
   DATA[812,33] := 0.3083624;
   DATA[812,34] := 2.0;
   DATA[812,35] := 250.5608;
   DATA[812,36] := 1.649953;
   DATA[812,37] := 189.3425;
   DATA[812,38] := 0.000128152;
   DATA[812,39] := 1.0;
   DATA[813,0] := 2.554527;
   DATA[813,1] := 565.3182;
   DATA[813,2] := 2.0;
   DATA[813,3] := 1.0;
   DATA[813,4] := 262.2404;
   DATA[813,5] := 8.46533;
   DATA[813,6] := 315.5601;
   DATA[813,8] := 1.0;
   DATA[813,9] := 1.0;
   DATA[813,10] := 1.0;
   DATA[813,11] := 2.032781;
   DATA[813,13] := 1010.758;
   DATA[813,14] := 1.0;
   DATA[813,15] := 1.0;
   DATA[813,16] := 1.0;
   DATA[813,17] := 1.0;
   DATA[813,18] := 1.0;
   DATA[813,19] := 1.0;
   DATA[813,20] := 148.808;
   DATA[813,21] := 155.7293;
   DATA[813,22] := 1.715439;
   DATA[813,23] := 972.5198;
   DATA[813,24] := 2.0;
   DATA[813,25] := 2.0;
   DATA[813,26] := 7.878942;
   DATA[813,27] := 144.7578;
   DATA[813,28] := 263.0415;
   DATA[813,29] := 11.84312;
   DATA[813,30] := 1.726993;
   DATA[813,31] := 1.289996;
   DATA[813,32] := 0.7352687;
   DATA[813,33] := 0.3083624;
   DATA[813,34] := 2.0;
   DATA[813,35] := 250.5608;
   DATA[813,36] := 1.746067;
   DATA[813,37] := 189.3425;
   DATA[813,38] := 0.000128152;
   DATA[813,39] := 1.0;
   DATA[814,0] := 2.55837;
   DATA[814,1] := 565.2004;
   DATA[814,2] := 2.0;
   DATA[814,3] := 1.0;
   DATA[814,4] := 262.2404;
   DATA[814,5] := 8.46533;
   DATA[814,6] := 315.3807;
   DATA[814,8] := 1.0;
   DATA[814,9] := 1.0;
   DATA[814,10] := 1.0;
   DATA[814,11] := 2.032781;
   DATA[814,13] := 1010.478;
   DATA[814,14] := 1.0;
   DATA[814,15] := 1.0;
   DATA[814,16] := 1.0;
   DATA[814,17] := 1.0;
   DATA[814,18] := 1.0;
   DATA[814,19] := 1.0;
   DATA[814,20] := 148.808;
   DATA[814,21] := 155.7293;
   DATA[814,22] := 1.715439;
   DATA[814,23] := 972.2507;
   DATA[814,24] := 2.0;
   DATA[814,25] := 2.0;
   DATA[814,26] := 7.878942;
   DATA[814,27] := 144.7578;
   DATA[814,28] := 263.0415;
   DATA[814,29] := 12.11228;
   DATA[814,30] := 1.726993;
   DATA[814,31] := 1.30178;
   DATA[814,32] := 0.7352687;
   DATA[814,33] := 0.3083624;
   DATA[814,34] := 2.0;
   DATA[814,35] := 250.5608;
   DATA[814,36] := 1.746067;
   DATA[814,37] := 189.3425;
   DATA[814,38] := 0.000128152;
   DATA[814,39] := 1.0;
   DATA[815,0] := 2.55837;
   DATA[815,1] := 564.8079;
   DATA[815,2] := 2.0;
   DATA[815,3] := 1.0;
   DATA[815,4] := 262.2404;
   DATA[815,5] := 8.46533;
   DATA[815,6] := 315.3807;
   DATA[815,8] := 1.0;
   DATA[815,9] := 1.0;
   DATA[815,10] := 1.0;
   DATA[815,11] := 2.032781;
   DATA[815,13] := 1010.638;
   DATA[815,14] := 1.0;
   DATA[815,15] := 1.0;
   DATA[815,16] := 1.0;
   DATA[815,17] := 1.0;
   DATA[815,18] := 1.0;
   DATA[815,19] := 1.0;
   DATA[815,20] := 148.808;
   DATA[815,21] := 155.7293;
   DATA[815,22] := 1.715439;
   DATA[815,23] := 972.1354;
   DATA[815,24] := 2.0;
   DATA[815,25] := 2.0;
   DATA[815,26] := 7.878942;
   DATA[815,27] := 144.7578;
   DATA[815,28] := 263.0415;
   DATA[815,29] := 12.11228;
   DATA[815,30] := 1.726993;
   DATA[815,31] := 1.30178;
   DATA[815,32] := 0.7352687;
   DATA[815,33] := 0.3083624;
   DATA[815,34] := 2.0;
   DATA[815,35] := 250.5608;
   DATA[815,36] := 1.746067;
   DATA[815,37] := 189.3425;
   DATA[815,38] := 0.000128152;
   DATA[815,39] := 1.0;
   DATA[816,0] := 2.55837;
   DATA[816,1] := 564.8472;
   DATA[816,2] := 2.0;
   DATA[816,3] := 1.0;
   DATA[816,4] := 262.2404;
   DATA[816,5] := 8.46533;
   DATA[816,6] := 315.3807;
   DATA[816,8] := 1.0;
   DATA[816,9] := 1.0;
   DATA[816,10] := 1.0;
   DATA[816,11] := 2.032781;
   DATA[816,13] := 1010.478;
   DATA[816,14] := 1.0;
   DATA[816,15] := 1.0;
   DATA[816,16] := 1.0;
   DATA[816,17] := 1.0;
   DATA[816,18] := 1.0;
   DATA[816,19] := 1.0;
   DATA[816,20] := 148.808;
   DATA[816,21] := 155.7293;
   DATA[816,22] := 1.715439;
   DATA[816,23] := 971.8662;
   DATA[816,24] := 2.0;
   DATA[816,25] := 2.0;
   DATA[816,26] := 7.878942;
   DATA[816,27] := 144.7578;
   DATA[816,28] := 263.0415;
   DATA[816,29] := 12.11228;
   DATA[816,30] := 1.726993;
   DATA[816,31] := 1.296401;
   DATA[816,32] := 0.7352687;
   DATA[816,33] := 0.3083624;
   DATA[816,34] := 2.0;
   DATA[816,35] := 250.5608;
   DATA[816,36] := 1.746067;
   DATA[816,37] := 189.3425;
   DATA[816,38] := 0.000128152;
   DATA[816,39] := 1.0;
   DATA[817,0] := 2.557089;
   DATA[817,1] := 564.6509;
   DATA[817,2] := 2.0;
   DATA[817,3] := 1.0;
   DATA[817,4] := 262.2404;
   DATA[817,5] := 8.46533;
   DATA[817,6] := 315.3807;
   DATA[817,8] := 1.0;
   DATA[817,9] := 1.0;
   DATA[817,10] := 1.0;
   DATA[817,11] := 2.032781;
   DATA[817,13] := 1010.638;
   DATA[817,14] := 1.0;
   DATA[817,15] := 1.0;
   DATA[817,16] := 1.0;
   DATA[817,17] := 1.0;
   DATA[817,18] := 1.0;
   DATA[817,19] := 1.0;
   DATA[817,20] := 148.808;
   DATA[817,21] := 155.7293;
   DATA[817,22] := 1.716721;
   DATA[817,23] := 971.4432;
   DATA[817,24] := 2.0;
   DATA[817,25] := 2.0;
   DATA[817,26] := 7.878942;
   DATA[817,27] := 144.7578;
   DATA[817,28] := 263.0415;
   DATA[817,29] := 12.11228;
   DATA[817,30] := 1.72507;
   DATA[817,31] := 1.291149;
   DATA[817,32] := 0.7352687;
   DATA[817,33] := 0.3083624;
   DATA[817,34] := 2.0;
   DATA[817,35] := 250.5608;
   DATA[817,36] := 1.746067;
   DATA[817,37] := 189.3425;
   DATA[817,38] := 0.000128152;
   DATA[817,39] := 1.0;
   DATA[818,0] := 2.548121;
   DATA[818,1] := 564.4547;
   DATA[818,2] := 2.0;
   DATA[818,3] := 1.0;
   DATA[818,4] := 262.2404;
   DATA[818,5] := 8.46533;
   DATA[818,6] := 315.3807;
   DATA[818,8] := 1.0;
   DATA[818,9] := 1.0;
   DATA[818,10] := 1.0;
   DATA[818,11] := 2.032781;
   DATA[818,13] := 1010.438;
   DATA[818,14] := 1.0;
   DATA[818,15] := 1.0;
   DATA[818,16] := 1.0;
   DATA[818,17] := 1.0;
   DATA[818,18] := 1.0;
   DATA[818,19] := 1.0;
   DATA[818,20] := 148.808;
   DATA[818,21] := 155.7293;
   DATA[818,22] := 1.717489;
   DATA[818,23] := 971.2894;
   DATA[818,24] := 2.0;
   DATA[818,25] := 2.0;
   DATA[818,26] := 7.878942;
   DATA[818,27] := 144.7578;
   DATA[818,28] := 263.0415;
   DATA[818,29] := 12.11228;
   DATA[818,30] := 1.72507;
   DATA[818,31] := 1.291149;
   DATA[818,32] := 0.7352687;
   DATA[818,33] := 0.3083624;
   DATA[818,34] := 2.0;
   DATA[818,35] := 250.5608;
   DATA[818,36] := 1.746067;
   DATA[818,37] := 189.3425;
   DATA[818,38] := 0.000128152;
   DATA[818,39] := 1.0;
   DATA[819,0] := 2.548121;
   DATA[819,1] := 565.2004;
   DATA[819,2] := 2.0;
   DATA[819,3] := 1.0;
   DATA[819,4] := 262.2404;
   DATA[819,5] := 8.46533;
   DATA[819,6] := 315.3807;
   DATA[819,8] := 1.0;
   DATA[819,9] := 1.0;
   DATA[819,10] := 1.0;
   DATA[819,11] := 2.032781;
   DATA[819,13] := 1010.558;
   DATA[819,14] := 1.0;
   DATA[819,15] := 1.0;
   DATA[819,16] := 1.0;
   DATA[819,17] := 1.0;
   DATA[819,18] := 1.0;
   DATA[819,19] := 1.0;
   DATA[819,20] := 148.808;
   DATA[819,21] := 155.7293;
   DATA[819,22] := 1.717489;
   DATA[819,23] := 970.7896;
   DATA[819,24] := 2.0;
   DATA[819,25] := 2.0;
   DATA[819,26] := 7.878942;
   DATA[819,27] := 144.7578;
   DATA[819,28] := 263.0415;
   DATA[819,29] := 12.11228;
   DATA[819,30] := 1.72507;
   DATA[819,31] := 1.291149;
   DATA[819,32] := 0.7352687;
   DATA[819,33] := 0.3083624;
   DATA[819,34] := 2.0;
   DATA[819,35] := 250.5608;
   DATA[819,36] := 1.746067;
   DATA[819,37] := 189.3425;
   DATA[819,38] := 0.000128152;
   DATA[819,39] := 1.0;
   DATA[820,0] := 2.543638;
   DATA[820,1] := 565.593;
   DATA[820,2] := 2.0;
   DATA[820,3] := 1.0;
   DATA[820,4] := 262.3366;
   DATA[820,5] := 8.46533;
   DATA[820,6] := 315.3807;
   DATA[820,8] := 1.0;
   DATA[820,9] := 1.0;
   DATA[820,10] := 1.0;
   DATA[820,11] := 2.032781;
   DATA[820,13] := 1010.438;
   DATA[820,14] := 1.0;
   DATA[820,15] := 1.0;
   DATA[820,16] := 1.0;
   DATA[820,17] := 1.0;
   DATA[820,18] := 1.0;
   DATA[820,19] := 1.0;
   DATA[820,20] := 148.808;
   DATA[820,21] := 155.7293;
   DATA[820,22] := 1.717489;
   DATA[820,23] := 970.5973;
   DATA[820,24] := 2.0;
   DATA[820,25] := 2.0;
   DATA[820,26] := 7.878942;
   DATA[820,27] := 144.7578;
   DATA[820,28] := 263.0415;
   DATA[820,29] := 12.11228;
   DATA[820,30] := 1.72507;
   DATA[820,31] := 1.291149;
   DATA[820,32] := 0.7352687;
   DATA[820,33] := 0.3083624;
   DATA[820,34] := 2.0;
   DATA[820,35] := 250.5608;
   DATA[820,36] := 1.730048;
   DATA[820,37] := 189.3425;
   DATA[820,38] := 0.000128152;
   DATA[820,39] := 1.0;
   DATA[821,0] := 2.543638;
   DATA[821,1] := 566.7706;
   DATA[821,2] := 2.0;
   DATA[821,3] := 1.0;
   DATA[821,4] := 262.3366;
   DATA[821,5] := 8.46533;
   DATA[821,6] := 315.3807;
   DATA[821,8] := 1.0;
   DATA[821,9] := 1.0;
   DATA[821,10] := 1.0;
   DATA[821,11] := 2.032781;
   DATA[821,13] := 1010.078;
   DATA[821,14] := 1.0;
   DATA[821,15] := 1.0;
   DATA[821,16] := 1.0;
   DATA[821,17] := 1.0;
   DATA[821,18] := 1.0;
   DATA[821,19] := 1.0;
   DATA[821,20] := 148.808;
   DATA[821,21] := 155.7037;
   DATA[821,22] := 1.717489;
   DATA[821,23] := 970.3666;
   DATA[821,24] := 2.0;
   DATA[821,25] := 2.0;
   DATA[821,26] := 7.878942;
   DATA[821,27] := 144.7578;
   DATA[821,28] := 263.0415;
   DATA[821,29] := 12.11228;
   DATA[821,30] := 1.72507;
   DATA[821,31] := 1.301652;
   DATA[821,32] := 0.7352687;
   DATA[821,33] := 0.3083624;
   DATA[821,34] := 2.0;
   DATA[821,35] := 250.5608;
   DATA[821,36] := 1.730048;
   DATA[821,37] := 189.3425;
   DATA[821,38] := 0.000128152;
   DATA[821,39] := 1.0;
   DATA[822,0] := 2.543638;
   DATA[822,1] := 567.3594;
   DATA[822,2] := 2.0;
   DATA[822,3] := 1.0;
   DATA[822,4] := 262.3366;
   DATA[822,5] := 8.46533;
   DATA[822,6] := 315.1243;
   DATA[822,8] := 1.0;
   DATA[822,9] := 1.0;
   DATA[822,10] := 1.0;
   DATA[822,11] := 2.032781;
   DATA[822,13] := 1010.118;
   DATA[822,14] := 1.0;
   DATA[822,15] := 1.0;
   DATA[822,16] := 1.0;
   DATA[822,17] := 1.0;
   DATA[822,18] := 1.0;
   DATA[822,19] := 1.0;
   DATA[822,20] := 148.808;
   DATA[822,21] := 155.6011;
   DATA[822,22] := 1.717489;
   DATA[822,23] := 970.1359;
   DATA[822,24] := 2.0;
   DATA[822,25] := 2.0;
   DATA[822,26] := 7.878942;
   DATA[822,27] := 144.7578;
   DATA[822,28] := 263.0415;
   DATA[822,29] := 12.11228;
   DATA[822,30] := 1.72507;
   DATA[822,31] := 1.29845;
   DATA[822,32] := 0.7352687;
   DATA[822,33] := 0.3083624;
   DATA[822,34] := 2.0;
   DATA[822,35] := 250.5608;
   DATA[822,36] := 1.730048;
   DATA[822,37] := 189.4066;
   DATA[822,38] := 0.000128152;
   DATA[822,39] := 1.0;
   DATA[823,0] := 2.542677;
   DATA[823,1] := 567.7911;
   DATA[823,2] := 2.0;
   DATA[823,3] := 1.0;
   DATA[823,4] := 262.3366;
   DATA[823,5] := 8.46533;
   DATA[823,6] := 315.1243;
   DATA[823,8] := 1.0;
   DATA[823,9] := 1.0;
   DATA[823,10] := 1.0;
   DATA[823,11] := 2.032781;
   DATA[823,13] := 1010.118;
   DATA[823,14] := 1.0;
   DATA[823,15] := 1.0;
   DATA[823,16] := 1.0;
   DATA[823,17] := 1.0;
   DATA[823,18] := 1.0;
   DATA[823,19] := 1.0;
   DATA[823,20] := 148.808;
   DATA[823,21] := 155.5755;
   DATA[823,22] := 1.717489;
   DATA[823,23] := 970.0205;
   DATA[823,24] := 2.0;
   DATA[823,25] := 2.0;
   DATA[823,26] := 7.878942;
   DATA[823,27] := 144.7578;
   DATA[823,28] := 263.0415;
   DATA[823,29] := 12.11228;
   DATA[823,30] := 1.72507;
   DATA[823,31] := 1.291918;
   DATA[823,32] := 0.7352687;
   DATA[823,33] := 0.3083624;
   DATA[823,34] := 2.0;
   DATA[823,35] := 250.5608;
   DATA[823,36] := 1.730048;
   DATA[823,37] := 189.4386;
   DATA[823,38] := 0.000128152;
   DATA[823,39] := 1.0;
   DATA[824,0] := 2.535311;
   DATA[824,1] := 568.1444;
   DATA[824,2] := 2.0;
   DATA[824,3] := 1.0;
   DATA[824,4] := 262.3366;
   DATA[824,5] := 8.46533;
   DATA[824,6] := 315.1243;
   DATA[824,8] := 1.0;
   DATA[824,9] := 1.0;
   DATA[824,10] := 1.0;
   DATA[824,11] := 2.032781;
   DATA[824,13] := 1010.118;
   DATA[824,14] := 1.0;
   DATA[824,15] := 1.0;
   DATA[824,16] := 1.0;
   DATA[824,17] := 1.0;
   DATA[824,18] := 1.0;
   DATA[824,19] := 1.0;
   DATA[824,20] := 148.808;
   DATA[824,21] := 155.5755;
   DATA[824,22] := 1.717489;
   DATA[824,23] := 970.0974;
   DATA[824,24] := 2.0;
   DATA[824,25] := 2.0;
   DATA[824,26] := 7.878942;
   DATA[824,27] := 144.7578;
   DATA[824,28] := 263.0415;
   DATA[824,29] := 12.11228;
   DATA[824,30] := 1.72507;
   DATA[824,31] := 1.291533;
   DATA[824,32] := 0.7352687;
   DATA[824,33] := 0.3083624;
   DATA[824,34] := 2.0;
   DATA[824,35] := 250.5768;
   DATA[824,36] := 1.730048;
   DATA[824,37] := 189.4386;
   DATA[824,38] := 0.000128152;
   DATA[824,39] := 1.0;
   DATA[825,0] := 2.535311;
   DATA[825,1] := 569.5575;
   DATA[825,2] := 2.0;
   DATA[825,3] := 1.0;
   DATA[825,4] := 262.3366;
   DATA[825,5] := 8.46533;
   DATA[825,6] := 315.1243;
   DATA[825,8] := 1.0;
   DATA[825,9] := 1.0;
   DATA[825,10] := 1.0;
   DATA[825,11] := 2.032781;
   DATA[825,13] := 1010.158;
   DATA[825,14] := 1.0;
   DATA[825,15] := 1.0;
   DATA[825,16] := 1.0;
   DATA[825,17] := 1.0;
   DATA[825,18] := 1.0;
   DATA[825,19] := 1.0;
   DATA[825,20] := 148.808;
   DATA[825,21] := 155.5755;
   DATA[825,22] := 1.717489;
   DATA[825,23] := 969.3668;
   DATA[825,24] := 2.0;
   DATA[825,25] := 2.0;
   DATA[825,26] := 7.878942;
   DATA[825,27] := 144.7578;
   DATA[825,28] := 263.0415;
   DATA[825,29] := 11.92002;
   DATA[825,30] := 1.72507;
   DATA[825,31] := 1.274881;
   DATA[825,32] := 0.7352687;
   DATA[825,33] := 0.3071454;
   DATA[825,34] := 2.0;
   DATA[825,35] := 250.721;
   DATA[825,36] := 1.730048;
   DATA[825,37] := 189.4386;
   DATA[825,38] := 0.000128152;
   DATA[825,39] := 1.0;
   DATA[826,0] := 2.544278;
   DATA[826,1] := 570.3426;
   DATA[826,2] := 2.0;
   DATA[826,3] := 1.0;
   DATA[826,4] := 262.3366;
   DATA[826,5] := 8.46533;
   DATA[826,6] := 315.1243;
   DATA[826,8] := 1.0;
   DATA[826,9] := 1.0;
   DATA[826,10] := 1.0;
   DATA[826,11] := 2.032781;
   DATA[826,13] := 1010.478;
   DATA[826,14] := 1.0;
   DATA[826,15] := 1.0;
   DATA[826,16] := 1.0;
   DATA[826,17] := 1.0;
   DATA[826,18] := 1.0;
   DATA[826,19] := 1.0;
   DATA[826,20] := 148.808;
   DATA[826,21] := 155.5755;
   DATA[826,22] := 1.717489;
   DATA[826,23] := 969.2515;
   DATA[826,24] := 2.0;
   DATA[826,25] := 2.0;
   DATA[826,26] := 7.878942;
   DATA[826,27] := 144.7578;
   DATA[826,28] := 263.0415;
   DATA[826,29] := 11.92002;
   DATA[826,30] := 1.72789;
   DATA[826,31] := 1.27898;
   DATA[826,32] := 0.7352687;
   DATA[826,33] := 0.3069532;
   DATA[826,34] := 2.0;
   DATA[826,35] := 250.721;
   DATA[826,36] := 1.730048;
   DATA[826,37] := 189.4386;
   DATA[826,38] := 0.000128152;
   DATA[826,39] := 1.0;
   DATA[827,0] := 2.547161;
   DATA[827,1] := 570.9706;
   DATA[827,2] := 2.0;
   DATA[827,3] := 1.0;
   DATA[827,4] := 262.3366;
   DATA[827,5] := 8.46533;
   DATA[827,6] := 315.1243;
   DATA[827,8] := 1.0;
   DATA[827,9] := 1.0;
   DATA[827,10] := 1.0;
   DATA[827,11] := 2.032781;
   DATA[827,13] := 1010.358;
   DATA[827,14] := 1.0;
   DATA[827,15] := 1.0;
   DATA[827,16] := 1.0;
   DATA[827,17] := 1.0;
   DATA[827,18] := 1.0;
   DATA[827,19] := 1.0;
   DATA[827,20] := 148.808;
   DATA[827,21] := 155.5755;
   DATA[827,22] := 1.719156;
   DATA[827,23] := 969.0208;
   DATA[827,24] := 2.0;
   DATA[827,25] := 2.0;
   DATA[827,26] := 7.878942;
   DATA[827,27] := 144.7578;
   DATA[827,28] := 263.0415;
   DATA[827,29] := 11.92002;
   DATA[827,30] := 1.728147;
   DATA[827,31] := 1.282183;
   DATA[827,32] := 0.7352687;
   DATA[827,33] := 0.3069532;
   DATA[827,34] := 2.0;
   DATA[827,35] := 250.721;
   DATA[827,36] := 1.730048;
   DATA[827,37] := 189.4386;
   DATA[827,38] := 0.000128152;
   DATA[827,39] := 1.0;
   DATA[828,0] := 2.547161;
   DATA[828,1] := 572.2659;
   DATA[828,2] := 2.0;
   DATA[828,3] := 1.0;
   DATA[828,4] := 262.3366;
   DATA[828,5] := 8.46533;
   DATA[828,6] := 315.1243;
   DATA[828,8] := 1.0;
   DATA[828,9] := 1.0;
   DATA[828,10] := 1.0;
   DATA[828,11] := 2.032781;
   DATA[828,13] := 1010.879;
   DATA[828,14] := 1.0;
   DATA[828,15] := 1.0;
   DATA[828,16] := 1.0;
   DATA[828,17] := 1.0;
   DATA[828,18] := 1.0;
   DATA[828,19] := 1.0;
   DATA[828,20] := 148.808;
   DATA[828,21] := 155.5755;
   DATA[828,22] := 1.719156;
   DATA[828,23] := 968.3671;
   DATA[828,24] := 2.0;
   DATA[828,25] := 2.0;
   DATA[828,26] := 7.878942;
   DATA[828,27] := 144.7578;
   DATA[828,28] := 263.0415;
   DATA[828,29] := 11.92002;
   DATA[828,30] := 1.728147;
   DATA[828,31] := 1.282183;
   DATA[828,32] := 0.7352687;
   DATA[828,33] := 0.3069532;
   DATA[828,34] := 2.0;
   DATA[828,35] := 250.721;
   DATA[828,36] := 1.730048;
   DATA[828,37] := 189.4386;
   DATA[828,38] := 0.000128152;
   DATA[828,39] := 1.0;
   DATA[829,0] := 2.547161;
   DATA[829,1] := 572.7762;
   DATA[829,2] := 2.0;
   DATA[829,3] := 1.0;
   DATA[829,4] := 262.3366;
   DATA[829,5] := 8.46533;
   DATA[829,6] := 315.1243;
   DATA[829,8] := 1.0;
   DATA[829,9] := 1.0;
   DATA[829,10] := 1.0;
   DATA[829,11] := 2.032781;
   DATA[829,13] := 1010.558;
   DATA[829,14] := 1.0;
   DATA[829,15] := 1.0;
   DATA[829,16] := 1.0;
   DATA[829,17] := 1.0;
   DATA[829,18] := 1.0;
   DATA[829,19] := 1.0;
   DATA[829,20] := 148.808;
   DATA[829,21] := 155.8062;
   DATA[829,22] := 1.719156;
   DATA[829,23] := 967.9056;
   DATA[829,24] := 2.0;
   DATA[829,25] := 2.0;
   DATA[829,26] := 7.878942;
   DATA[829,27] := 144.7578;
   DATA[829,28] := 263.0415;
   DATA[829,29] := 11.92002;
   DATA[829,30] := 1.729557;
   DATA[829,31] := 1.282183;
   DATA[829,32] := 0.7352687;
   DATA[829,33] := 0.3065689;
   DATA[829,34] := 2.0;
   DATA[829,35] := 250.721;
   DATA[829,36] := 1.730048;
   DATA[829,37] := 189.4386;
   DATA[829,38] := 0.000128152;
   DATA[829,39] := 1.0;
   DATA[830,0] := 2.547161;
   DATA[830,1] := 573.2473;
   DATA[830,2] := 2.0;
   DATA[830,3] := 1.0;
   DATA[830,4] := 262.3366;
   DATA[830,5] := 8.46533;
   DATA[830,6] := 315.1243;
   DATA[830,8] := 1.0;
   DATA[830,9] := 1.0;
   DATA[830,10] := 1.0;
   DATA[830,11] := 2.032781;
   DATA[830,13] := 1010.919;
   DATA[830,14] := 1.0;
   DATA[830,15] := 1.0;
   DATA[830,16] := 1.0;
   DATA[830,17] := 1.0;
   DATA[830,18] := 1.0;
   DATA[830,19] := 1.0;
   DATA[830,20] := 148.808;
   DATA[830,21] := 155.8062;
   DATA[830,22] := 1.717746;
   DATA[830,23] := 967.4827;
   DATA[830,24] := 2.0;
   DATA[830,25] := 2.0;
   DATA[830,26] := 7.878942;
   DATA[830,27] := 144.7578;
   DATA[830,28] := 263.0415;
   DATA[830,29] := 11.92002;
   DATA[830,30] := 1.729557;
   DATA[830,31] := 1.282183;
   DATA[830,32] := 0.7352687;
   DATA[830,33] := 0.3079781;
   DATA[830,34] := 2.0;
   DATA[830,35] := 250.4967;
   DATA[830,36] := 1.730048;
   DATA[830,37] := 189.4386;
   DATA[830,38] := 0.000128152;
   DATA[830,39] := 1.0;
   DATA[831,0] := 2.547161;
   DATA[831,1] := 573.3258;
   DATA[831,2] := 2.0;
   DATA[831,3] := 1.0;
   DATA[831,4] := 262.3366;
   DATA[831,5] := 8.46533;
   DATA[831,6] := 315.1243;
   DATA[831,8] := 1.0;
   DATA[831,9] := 1.0;
   DATA[831,10] := 1.0;
   DATA[831,11] := 2.032781;
   DATA[831,13] := 1010.718;
   DATA[831,14] := 1.0;
   DATA[831,15] := 1.0;
   DATA[831,16] := 1.0;
   DATA[831,17] := 1.0;
   DATA[831,18] := 1.0;
   DATA[831,19] := 1.0;
   DATA[831,20] := 148.808;
   DATA[831,21] := 155.8062;
   DATA[831,22] := 1.717746;
   DATA[831,23] := 967.3289;
   DATA[831,24] := 2.0;
   DATA[831,25] := 2.0;
   DATA[831,26] := 7.878942;
   DATA[831,27] := 144.7578;
   DATA[831,28] := 263.0415;
   DATA[831,29] := 11.92002;
   DATA[831,30] := 1.729557;
   DATA[831,31] := 1.271935;
   DATA[831,32] := 0.7352687;
   DATA[831,33] := 0.3083624;
   DATA[831,34] := 2.0;
   DATA[831,35] := 250.4967;
   DATA[831,36] := 1.730048;
   DATA[831,37] := 189.4386;
   DATA[831,38] := 0.000128152;
   DATA[831,39] := 1.0;
   DATA[832,0] := 2.547161;
   DATA[832,1] := 574.4249;
   DATA[832,2] := 2.0;
   DATA[832,3] := 1.0;
   DATA[832,4] := 262.3366;
   DATA[832,5] := 8.46533;
   DATA[832,6] := 315.1243;
   DATA[832,8] := 1.0;
   DATA[832,9] := 1.0;
   DATA[832,10] := 1.0;
   DATA[832,11] := 2.032781;
   DATA[832,13] := 1011.039;
   DATA[832,14] := 1.0;
   DATA[832,15] := 1.0;
   DATA[832,16] := 1.0;
   DATA[832,17] := 1.0;
   DATA[832,18] := 1.0;
   DATA[832,19] := 1.0;
   DATA[832,20] := 148.808;
   DATA[832,21] := 155.5755;
   DATA[832,22] := 1.717746;
   DATA[832,23] := 966.9059;
   DATA[832,24] := 2.0;
   DATA[832,25] := 2.0;
   DATA[832,26] := 7.878942;
   DATA[832,27] := 144.7578;
   DATA[832,28] := 263.0415;
   DATA[832,29] := 11.92002;
   DATA[832,30] := 1.729557;
   DATA[832,31] := 1.279621;
   DATA[832,32] := 0.7352687;
   DATA[832,33] := 0.3083624;
   DATA[832,34] := 2.0;
   DATA[832,35] := 250.4967;
   DATA[832,36] := 1.730048;
   DATA[832,37] := 189.4386;
   DATA[832,38] := 0.000128152;
   DATA[832,39] := 1.0;
   DATA[833,0] := 2.555168;
   DATA[833,1] := 575.4454;
   DATA[833,2] := 2.0;
   DATA[833,3] := 1.0;
   DATA[833,4] := 262.3366;
   DATA[833,5] := 8.46533;
   DATA[833,6] := 315.1243;
   DATA[833,8] := 1.0;
   DATA[833,9] := 1.0;
   DATA[833,10] := 1.0;
   DATA[833,11] := 2.032781;
   DATA[833,13] := 1010.959;
   DATA[833,14] := 1.0;
   DATA[833,15] := 1.0;
   DATA[833,16] := 1.0;
   DATA[833,17] := 1.0;
   DATA[833,18] := 1.0;
   DATA[833,19] := 1.0;
   DATA[833,20] := 148.808;
   DATA[833,21] := 155.5755;
   DATA[833,22] := 1.717746;
   DATA[833,23] := 966.6752;
   DATA[833,24] := 2.0;
   DATA[833,25] := 2.0;
   DATA[833,26] := 7.878942;
   DATA[833,27] := 144.7578;
   DATA[833,28] := 263.0415;
   DATA[833,29] := 12.15073;
   DATA[833,30] := 1.729557;
   DATA[833,31] := 1.290893;
   DATA[833,32] := 0.7352687;
   DATA[833,33] := 0.3083624;
   DATA[833,34] := 2.0;
   DATA[833,35] := 250.737;
   DATA[833,36] := 1.730048;
   DATA[833,37] := 189.4386;
   DATA[833,38] := 0.000128152;
   DATA[833,39] := 1.0;
   DATA[834,0] := 2.555168;
   DATA[834,1] := 576.2697;
   DATA[834,2] := 2.0;
   DATA[834,3] := 1.0;
   DATA[834,4] := 262.3366;
   DATA[834,5] := 8.46533;
   DATA[834,6] := 315.1243;
   DATA[834,8] := 1.0;
   DATA[834,9] := 1.0;
   DATA[834,10] := 1.0;
   DATA[834,11] := 2.032781;
   DATA[834,13] := 1011.279;
   DATA[834,14] := 1.0;
   DATA[834,15] := 1.0;
   DATA[834,16] := 1.0;
   DATA[834,17] := 1.0;
   DATA[834,18] := 1.0;
   DATA[834,19] := 1.0;
   DATA[834,20] := 148.808;
   DATA[834,21] := 155.5755;
   DATA[834,22] := 1.717746;
   DATA[834,23] := 966.3676;
   DATA[834,24] := 2.0;
   DATA[834,25] := 2.0;
   DATA[834,26] := 7.878942;
   DATA[834,27] := 144.7578;
   DATA[834,28] := 263.0415;
   DATA[834,29] := 12.15073;
   DATA[834,30] := 1.729557;
   DATA[834,31] := 1.286153;
   DATA[834,32] := 0.7352687;
   DATA[834,33] := 0.3083624;
   DATA[834,34] := 2.0;
   DATA[834,35] := 250.737;
   DATA[834,36] := 1.730048;
   DATA[834,37] := 189.4386;
   DATA[834,38] := 0.000128152;
   DATA[834,39] := 1.0;
   DATA[835,0] := 2.555168;
   DATA[835,1] := 577.251;
   DATA[835,2] := 2.0;
   DATA[835,3] := 1.0;
   DATA[835,4] := 262.3366;
   DATA[835,5] := 8.46533;
   DATA[835,6] := 315.1243;
   DATA[835,8] := 1.0;
   DATA[835,9] := 1.0;
   DATA[835,10] := 1.0;
   DATA[835,11] := 2.032781;
   DATA[835,13] := 1011.079;
   DATA[835,14] := 1.0;
   DATA[835,15] := 1.0;
   DATA[835,16] := 1.0;
   DATA[835,17] := 1.0;
   DATA[835,18] := 1.0;
   DATA[835,19] := 1.0;
   DATA[835,20] := 148.808;
   DATA[835,21] := 155.5755;
   DATA[835,22] := 1.717746;
   DATA[835,23] := 965.7139;
   DATA[835,24] := 2.0;
   DATA[835,25] := 2.0;
   DATA[835,26] := 7.878942;
   DATA[835,27] := 144.7578;
   DATA[835,28] := 263.0415;
   DATA[835,29] := 12.15073;
   DATA[835,30] := 1.7293;
   DATA[835,31] := 1.288715;
   DATA[835,32] := 0.7352687;
   DATA[835,33] := 0.3083624;
   DATA[835,34] := 2.0;
   DATA[835,35] := 250.737;
   DATA[835,36] := 1.730048;
   DATA[835,37] := 189.6949;
   DATA[835,38] := 0.000128152;
   DATA[835,39] := 1.0;
   DATA[836,0] := 2.555168;
   DATA[836,1] := 577.8006;
   DATA[836,2] := 2.0;
   DATA[836,3] := 1.0;
   DATA[836,4] := 262.3366;
   DATA[836,5] := 8.46533;
   DATA[836,6] := 315.1243;
   DATA[836,8] := 1.0;
   DATA[836,9] := 1.0;
   DATA[836,10] := 1.0;
   DATA[836,11] := 2.032781;
   DATA[836,13] := 1011.079;
   DATA[836,14] := 1.0;
   DATA[836,15] := 1.0;
   DATA[836,16] := 1.0;
   DATA[836,17] := 1.0;
   DATA[836,18] := 1.0;
   DATA[836,19] := 1.0;
   DATA[836,20] := 148.808;
   DATA[836,21] := 155.5755;
   DATA[836,22] := 1.718515;
   DATA[836,23] := 965.3294;
   DATA[836,24] := 2.0;
   DATA[836,25] := 2.0;
   DATA[836,26] := 7.878942;
   DATA[836,27] := 144.7578;
   DATA[836,28] := 263.0415;
   DATA[836,29] := 12.15073;
   DATA[836,30] := 1.7293;
   DATA[836,31] := 1.281542;
   DATA[836,32] := 0.7352687;
   DATA[836,33] := 0.3083624;
   DATA[836,34] := 2.0;
   DATA[836,35] := 250.8972;
   DATA[836,36] := 1.730048;
   DATA[836,37] := 189.6949;
   DATA[836,38] := 0.000128152;
   DATA[836,39] := 1.0;
   DATA[837,0] := 2.555168;
   DATA[837,1] := 578.8212;
   DATA[837,2] := 2.0;
   DATA[837,3] := 1.0;
   DATA[837,4] := 262.3366;
   DATA[837,5] := 8.46533;
   DATA[837,6] := 315.1243;
   DATA[837,8] := 1.0;
   DATA[837,9] := 1.0;
   DATA[837,10] := 1.0;
   DATA[837,11] := 2.032781;
   DATA[837,13] := 1011.239;
   DATA[837,14] := 1.0;
   DATA[837,15] := 1.0;
   DATA[837,16] := 1.0;
   DATA[837,17] := 1.0;
   DATA[837,18] := 1.0;
   DATA[837,19] := 1.0;
   DATA[837,20] := 148.808;
   DATA[837,21] := 155.5755;
   DATA[837,22] := 1.720565;
   DATA[837,23] := 964.6373;
   DATA[837,24] := 2.0;
   DATA[837,25] := 2.0;
   DATA[837,26] := 7.878942;
   DATA[837,27] := 144.7578;
   DATA[837,28] := 263.0415;
   DATA[837,29] := 12.15073;
   DATA[837,30] := 1.7293;
   DATA[837,31] := 1.272192;
   DATA[837,32] := 0.7352687;
   DATA[837,33] := 0.3083624;
   DATA[837,34] := 2.0;
   DATA[837,35] := 250.8972;
   DATA[837,36] := 1.730048;
   DATA[837,37] := 189.6949;
   DATA[837,38] := 0.000128152;
   DATA[837,39] := 1.0;
   DATA[838,0] := 2.553886;
   DATA[838,1] := 579.724;
   DATA[838,2] := 2.0;
   DATA[838,3] := 1.0;
   DATA[838,4] := 262.3366;
   DATA[838,5] := 8.46533;
   DATA[838,6] := 315.1243;
   DATA[838,8] := 1.0;
   DATA[838,9] := 1.0;
   DATA[838,10] := 1.0;
   DATA[838,11] := 2.032781;
   DATA[838,13] := 1011.279;
   DATA[838,14] := 1.0;
   DATA[838,15] := 1.0;
   DATA[838,16] := 1.0;
   DATA[838,17] := 1.0;
   DATA[838,18] := 1.0;
   DATA[838,19] := 1.0;
   DATA[838,20] := 148.808;
   DATA[838,21] := 155.5755;
   DATA[838,22] := 1.720565;
   DATA[838,23] := 964.5988;
   DATA[838,24] := 2.0;
   DATA[838,25] := 2.0;
   DATA[838,26] := 7.878942;
   DATA[838,27] := 144.7578;
   DATA[838,28] := 263.0415;
   DATA[838,29] := 12.15073;
   DATA[838,30] := 1.7293;
   DATA[838,31] := 1.271679;
   DATA[838,32] := 0.736421;
   DATA[838,33] := 0.3083624;
   DATA[838,34] := 2.0;
   DATA[838,35] := 250.8972;
   DATA[838,36] := 1.730048;
   DATA[838,37] := 189.6949;
   DATA[838,38] := 0.000128152;
   DATA[838,39] := 1.0;
   DATA[839,0] := 2.54684;
   DATA[839,1] := 580.7053;
   DATA[839,2] := 2.0;
   DATA[839,3] := 1.0;
   DATA[839,4] := 262.3366;
   DATA[839,5] := 8.46533;
   DATA[839,6] := 315.1243;
   DATA[839,8] := 1.0;
   DATA[839,9] := 1.0;
   DATA[839,10] := 1.0;
   DATA[839,11] := 2.032781;
   DATA[839,13] := 1011.079;
   DATA[839,14] := 1.0;
   DATA[839,15] := 1.0;
   DATA[839,16] := 1.0;
   DATA[839,17] := 1.0;
   DATA[839,18] := 1.0;
   DATA[839,19] := 1.0;
   DATA[839,20] := 148.808;
   DATA[839,21] := 155.5755;
   DATA[839,22] := 1.720565;
   DATA[839,23] := 964.1758;
   DATA[839,24] := 2.0;
   DATA[839,25] := 2.0;
   DATA[839,26] := 7.878942;
   DATA[839,27] := 144.7578;
   DATA[839,28] := 263.0415;
   DATA[839,29] := 12.15073;
   DATA[839,30] := 1.7293;
   DATA[839,31] := 1.271551;
   DATA[839,32] := 0.7366771;
   DATA[839,33] := 0.3068891;
   DATA[839,34] := 2.0;
   DATA[839,35] := 250.8972;
   DATA[839,36] := 1.730048;
   DATA[839,37] := 189.5668;
   DATA[839,38] := 0.000128152;
   DATA[839,39] := 1.0;
   DATA[840,0] := 2.542356;
   DATA[840,1] := 581.2941;
   DATA[840,2] := 2.0;
   DATA[840,3] := 1.0;
   DATA[840,4] := 262.3366;
   DATA[840,5] := 8.46533;
   DATA[840,6] := 315.1243;
   DATA[840,8] := 1.0;
   DATA[840,9] := 1.0;
   DATA[840,10] := 1.0;
   DATA[840,11] := 2.026378;
   DATA[840,13] := 1010.879;
   DATA[840,14] := 1.0;
   DATA[840,15] := 1.0;
   DATA[840,16] := 1.0;
   DATA[840,17] := 1.0;
   DATA[840,18] := 1.0;
   DATA[840,19] := 1.0;
   DATA[840,20] := 148.808;
   DATA[840,21] := 155.5755;
   DATA[840,22] := 1.718771;
   DATA[840,23] := 963.7529;
   DATA[840,24] := 2.0;
   DATA[840,25] := 2.0;
   DATA[840,26] := 7.878942;
   DATA[840,27] := 144.7578;
   DATA[840,28] := 263.0415;
   DATA[840,29] := 12.15073;
   DATA[840,30] := 1.728019;
   DATA[840,31] := 1.271551;
   DATA[840,32] := 0.7373172;
   DATA[840,33] := 0.3068891;
   DATA[840,34] := 2.0;
   DATA[840,35] := 250.785;
   DATA[840,36] := 1.730048;
   DATA[840,37] := 189.4546;
   DATA[840,38] := 0.000128152;
   DATA[840,39] := 1.0;
   DATA[841,0] := 2.538833;
   DATA[841,1] := 581.5688;
   DATA[841,2] := 2.0;
   DATA[841,3] := 1.0;
   DATA[841,4] := 262.3366;
   DATA[841,5] := 8.46501;
   DATA[841,6] := 315.1243;
   DATA[841,8] := 1.0;
   DATA[841,9] := 1.0;
   DATA[841,10] := 1.0;
   DATA[841,11] := 2.026378;
   DATA[841,13] := 1011.159;
   DATA[841,14] := 1.0;
   DATA[841,15] := 1.0;
   DATA[841,16] := 1.0;
   DATA[841,17] := 1.0;
   DATA[841,18] := 1.0;
   DATA[841,19] := 1.0;
   DATA[841,20] := 148.808;
   DATA[841,21] := 155.5755;
   DATA[841,22] := 1.718771;
   DATA[841,23] := 963.4068;
   DATA[841,24] := 2.0;
   DATA[841,25] := 2.0;
   DATA[841,26] := 7.878942;
   DATA[841,27] := 144.7578;
   DATA[841,28] := 263.0415;
   DATA[841,29] := 12.15073;
   DATA[841,30] := 1.726609;
   DATA[841,31] := 1.271551;
   DATA[841,32] := 0.7383414;
   DATA[841,33] := 0.3068891;
   DATA[841,34] := 2.0;
   DATA[841,35] := 250.4807;
   DATA[841,36] := 1.730048;
   DATA[841,37] := 189.1983;
   DATA[841,38] := 0.000128152;
   DATA[841,39] := 1.0;
   DATA[842,0] := 2.538833;
   DATA[842,1] := 581.5688;
   DATA[842,2] := 2.0;
   DATA[842,3] := 1.0;
   DATA[842,4] := 262.3366;
   DATA[842,5] := 8.46501;
   DATA[842,6] := 315.1243;
   DATA[842,8] := 1.0;
   DATA[842,9] := 1.0;
   DATA[842,10] := 1.0;
   DATA[842,11] := 2.026378;
   DATA[842,13] := 1011.159;
   DATA[842,14] := 1.0;
   DATA[842,15] := 1.0;
   DATA[842,16] := 1.0;
   DATA[842,17] := 1.0;
   DATA[842,18] := 1.0;
   DATA[842,19] := 1.0;
   DATA[842,20] := 148.808;
   DATA[842,21] := 155.5755;
   DATA[842,22] := 1.718771;
   DATA[842,23] := 963.4068;
   DATA[842,24] := 2.0;
   DATA[842,25] := 2.0;
   DATA[842,26] := 7.878942;
   DATA[842,27] := 144.7578;
   DATA[842,28] := 263.0415;
   DATA[842,29] := 12.15073;
   DATA[842,30] := 1.726609;
   DATA[842,31] := 1.271551;
   DATA[842,32] := 0.7383414;
   DATA[842,33] := 0.3068891;
   DATA[842,34] := 2.0;
   DATA[842,35] := 250.4807;
   DATA[842,36] := 1.730048;
   DATA[842,37] := 189.1983;
   DATA[842,38] := 0.000128152;
   DATA[842,39] := 1.0;
   DATA[843,0] := 2.536912;
   DATA[843,1] := 581.9614;
   DATA[843,2] := 2.0;
   DATA[843,3] := 1.0;
   DATA[843,4] := 262.3366;
   DATA[843,5] := 8.462446;
   DATA[843,6] := 315.1243;
   DATA[843,8] := 1.0;
   DATA[843,9] := 1.0;
   DATA[843,10] := 1.0;
   DATA[843,11] := 2.026378;
   DATA[843,13] := 1011.039;
   DATA[843,14] := 1.0;
   DATA[843,15] := 1.0;
   DATA[843,16] := 1.0;
   DATA[843,17] := 1.0;
   DATA[843,18] := 1.0;
   DATA[843,19] := 1.0;
   DATA[843,20] := 148.808;
   DATA[843,21] := 155.5499;
   DATA[843,22] := 1.718771;
   DATA[843,23] := 963.2914;
   DATA[843,24] := 2.0;
   DATA[843,25] := 2.0;
   DATA[843,26] := 7.878942;
   DATA[843,27] := 144.7578;
   DATA[843,28] := 263.0415;
   DATA[843,29] := 12.15073;
   DATA[843,30] := 1.726609;
   DATA[843,31] := 1.281158;
   DATA[843,32] := 0.7368051;
   DATA[843,33] := 0.3068891;
   DATA[843,34] := 2.0;
   DATA[843,35] := 250.4807;
   DATA[843,36] := 1.730048;
   DATA[843,37] := 189.1983;
   DATA[843,38] := 0.000128152;
   DATA[843,39] := 1.0;
   DATA[844,0] := 2.544278;
   DATA[844,1] := 582.1577;
   DATA[844,2] := 2.0;
   DATA[844,3] := 1.0;
   DATA[844,4] := 262.3366;
   DATA[844,5] := 8.462446;
   DATA[844,6] := 315.1243;
   DATA[844,8] := 1.0;
   DATA[844,9] := 1.0;
   DATA[844,10] := 1.0;
   DATA[844,11] := 2.026378;
   DATA[844,13] := 1011.359;
   DATA[844,14] := 1.0;
   DATA[844,15] := 1.0;
   DATA[844,16] := 1.0;
   DATA[844,17] := 1.0;
   DATA[844,18] := 1.0;
   DATA[844,19] := 1.0;
   DATA[844,20] := 148.808;
